gfCNCPoint4[25196] = {X 2.3034, Y 2.3049, Z -6.3333, A 0.000, B 0.000, C 0.000 }
gfCNCPoint4[25197] = {X 2.3034, Y 6.8597, Z -6.3333, A 0.000, B 0.000, C 0.000 }
gfCNCPoint4[25198] = {X 2.4167, Y 6.8824, Z -6.3333, A 0.000, B 0.000, C 0.000 }
gfCNCPoint4[25199] = {X 4.7221, Y 6.0045, Z -6.3333, A 0.000, B 0.000, C 0.000 }
gfCNCPoint4[25200] = {X 7.0996, Y 5.3466, Z -6.3333, A 0.000, B 0.000, C 0.000 }
gfCNCPoint4[25201] = {X 9.5283, Y 4.9145, Z -6.3333, A 0.000, B 0.000, C 0.000 }
gfCNCPoint4[25202] = {X 11.9868, Y 4.7120, Z -6.3333, A 0.000, B 0.000, C 0.000 }
gfCNCPoint4[25203] = {X 14.4535, Y 4.7409, Z -6.3333, A 0.000, B 0.000, C 0.000 }
gfCNCPoint4[25204] = {X 16.9066, Y 5.0009, Z -6.3333, A 0.000, B 0.000, C 0.000 }
gfCNCPoint4[25205] = {X 18.9210, Y 5.4155, Z -6.3333, A 0.000, B 0.000, C 0.000 }
gfCNCPoint4[25206] = {X 20.8820, Y 6.0355, Z -6.3333, A 0.000, B 0.000, C 0.000 }
gfCNCPoint4[25207] = {X 22.7686, Y 6.8543, Z -6.3333, A 0.000, B 0.000, C 0.000 }
gfCNCPoint4[25208] = {X 24.4892, Y 7.8180, Z -6.3333, A 0.000, B 0.000, C 0.000 }
gfCNCPoint4[25209] = {X 26.1061, Y 8.9471, Z -6.3333, A 0.000, B 0.000, C 0.000 }
gfCNCPoint4[25210] = {X 27.4004, Y 10.0775, Z -6.3333, A 0.000, B 0.000, C 0.000 }
gfCNCPoint4[25211] = {X 28.5615, Y 11.3443, Z -6.3333, A 0.000, B 0.000, C 0.000 }
gfCNCPoint4[25212] = {X 29.5750, Y 12.7320, Z -6.3333, A 0.000, B 0.000, C 0.000 }
gfCNCPoint4[25213] = {X 30.4284, Y 14.2234, Z -6.3333, A 0.000, B 0.000, C 0.000 }
gfCNCPoint4[25214] = {X 31.1113, Y 15.8003, Z -6.3333, A 0.000, B 0.000, C 0.000 }
gfCNCPoint4[25215] = {X 31.6710, Y 17.7360, Z -6.3333, A 0.000, B 0.000, C 0.000 }
gfCNCPoint4[25216] = {X 32.0043, Y 19.7232, Z -6.3333, A 0.000, B 0.000, C 0.000 }
gfCNCPoint4[25217] = {X 32.1066, Y 21.7356, Z -6.3333, A 0.000, B 0.000, C 0.000 }
gfCNCPoint4[25218] = {X 31.9766, Y 23.7463, Z -6.3333, A 0.000, B 0.000, C 0.000 }
gfCNCPoint4[25219] = {X 31.6161, Y 25.7288, Z -6.3333, A 0.000, B 0.000, C 0.000 }
gfCNCPoint4[25220] = {X 31.1971, Y 27.1578, Z -6.3333, A 0.000, B 0.000, C 0.000 }
gfCNCPoint4[25221] = {X 30.6305, Y 28.5350, Z -6.3333, A 0.000, B 0.000, C 0.000 }
gfCNCPoint4[25222] = {X 29.9224, Y 29.8451, Z -6.3333, A 0.000, B 0.000, C 0.000 }
gfCNCPoint4[25223] = {X 29.0809, Y 31.0736, Z -6.3333, A 0.000, B 0.000, C 0.000 }
gfCNCPoint4[25224] = {X 29.6386, Y 31.7921, Z -6.3333, A 0.000, B 0.000, C 0.000 }
gfCNCPoint4[25225] = {X 30.0955, Y 32.5786, Z -6.3333, A 0.000, B 0.000, C 0.000 }
gfCNCPoint4[25226] = {X 33.1423, Y 38.8726, Z -6.3333, A 0.000, B 0.000, C 0.000 }
gfCNCPoint4[25227] = {X 33.5391, Y 39.8957, Z -6.3333, A 0.000, B 0.000, C 0.000 }
gfCNCPoint4[25228] = {X 33.7662, Y 40.9694, Z -6.3333, A 0.000, B 0.000, C 0.000 }
gfCNCPoint4[25229] = {X 33.8177, Y 42.0656, Z -6.3333, A 0.000, B 0.000, C 0.000 }
gfCNCPoint4[25230] = {X 33.7164, Y 43.0266, Z -6.3333, A 0.000, B 0.000, C 0.000 }
gfCNCPoint4[25231] = {X 33.4799, Y 43.9636, Z -6.3333, A 0.000, B 0.000, C 0.000 }
gfCNCPoint4[25232] = {X 33.1103, Y 44.8630, Z -6.3333, A 0.000, B 0.000, C 0.000 }
gfCNCPoint4[25233] = {X 32.6161, Y 45.7005, Z -6.3333, A 0.000, B 0.000, C 0.000 }
gfCNCPoint4[25234] = {X 32.0075, Y 46.4590, Z -6.3333, A 0.000, B 0.000, C 0.000 }
gfCNCPoint4[25235] = {X 31.2970, Y 47.1229, Z -6.3333, A 0.000, B 0.000, C 0.000 }
gfCNCPoint4[25236] = {X 30.7609, Y 47.5564, Z -6.3333, A 0.000, B 0.000, C 0.000 }
gfCNCPoint4[25237] = {X 29.8550, Y 48.1752, Z -6.3333, A 0.000, B 0.000, C 0.000 }
gfCNCPoint4[25238] = {X 28.8614, Y 48.6406, Z -6.3333, A 0.000, B 0.000, C 0.000 }
gfCNCPoint4[25239] = {X 27.8061, Y 48.9404, Z -6.3333, A 0.000, B 0.000, C 0.000 }
gfCNCPoint4[25240] = {X 26.7162, Y 49.0669, Z -6.3333, A 0.000, B 0.000, C 0.000 }
gfCNCPoint4[25241] = {X 25.6202, Y 49.0168, Z -6.3333, A 0.000, B 0.000, C 0.000 }
gfCNCPoint4[25242] = {X 23.9293, Y 49.8556, Z -6.3333, A 0.000, B 0.000, C 0.000 }
gfCNCPoint4[25243] = {X 22.1916, Y 50.5926, Z -6.3333, A 0.000, B 0.000, C 0.000 }
gfCNCPoint4[25244] = {X 20.4133, Y 51.2255, Z -6.3333, A 0.000, B 0.000, C 0.000 }
gfCNCPoint4[25245] = {X 18.2641, Y 51.8314, Z -6.3333, A 0.000, B 0.000, C 0.000 }
gfCNCPoint4[25246] = {X 16.0697, Y 52.2450, Z -6.3333, A 0.000, B 0.000, C 0.000 }
gfCNCPoint4[25247] = {X 13.8474, Y 52.4629, Z -6.3333, A 0.000, B 0.000, C 0.000 }
gfCNCPoint4[25248] = {X 11.6145, Y 52.4835, Z -6.3333, A 0.000, B 0.000, C 0.000 }
gfCNCPoint4[25249] = {X 9.3885, Y 52.3066, Z -6.3333, A 0.000, B 0.000, C 0.000 }
gfCNCPoint4[25250] = {X 7.1868, Y 51.9336, Z -6.3333, A 0.000, B 0.000, C 0.000 }
gfCNCPoint4[25251] = {X 6.2986, Y 51.7232, Z -6.3333, A 0.000, B 0.000, C 0.000 }
gfCNCPoint4[25252] = {X 5.4214, Y 51.4709, Z -6.3333, A 0.000, B 0.000, C 0.000 }
gfCNCPoint4[25253] = {X 3.8340, Y 50.8954, Z -6.3333, A 0.000, B 0.000, C 0.000 }
gfCNCPoint4[25254] = {X 2.3034, Y 50.1826, Z -6.3333, A 0.000, B 0.000, C 0.000 }
gfCNCPoint4[25255] = {X 2.3034, Y 97.6951, Z -6.3333, A 0.000, B 0.000, C 0.000 }
gfCNCPoint4[25256] = {X 120.1200, Y 97.6951, Z -6.3333, A 0.000, B 0.000, C 0.000 }
gfCNCPoint4[25257] = {X 120.1200, Y 97.0659, Z -6.3333, A 0.000, B 0.000, C 0.000 }
gfCNCPoint4[25258] = {X 120.2337, Y 96.0185, Z -6.3333, A 0.000, B 0.000, C 0.000 }
gfCNCPoint4[25259] = {X 120.5696, Y 95.0199, Z -6.3333, A 0.000, B 0.000, C 0.000 }
gfCNCPoint4[25260] = {X 121.1121, Y 94.1166, Z -6.3333, A 0.000, B 0.000, C 0.000 }
gfCNCPoint4[25261] = {X 121.8357, Y 93.3509, Z -6.3333, A 0.000, B 0.000, C 0.000 }
gfCNCPoint4[25262] = {X 122.7069, Y 92.7583, Z -6.3333, A 0.000, B 0.000, C 0.000 }
gfCNCPoint4[25263] = {X 123.6849, Y 92.3665, Z -6.3333, A 0.000, B 0.000, C 0.000 }
gfCNCPoint4[25264] = {X 124.7243, Y 92.1937, Z -6.3333, A 0.000, B 0.000, C 0.000 }
gfCNCPoint4[25265] = {X 124.7845, Y 92.1782, Z -6.3333, A 0.000, B 0.000, C 0.000 }
gfCNCPoint4[25266] = {X 124.8456, Y 92.1669, Z -6.3333, A 0.000, B 0.000, C 0.000 }
gfCNCPoint4[25267] = {X 125.3649, Y 92.0898, Z -6.3333, A 0.000, B 0.000, C 0.000 }
gfCNCPoint4[25268] = {X 126.0997, Y 91.9688, Z -6.3333, A 0.000, B 0.000, C 0.000 }
gfCNCPoint4[25269] = {X 126.8253, Y 91.8014, Z -6.3333, A 0.000, B 0.000, C 0.000 }
gfCNCPoint4[25270] = {X 127.9746, Y 90.7110, Z -6.3333, A 0.000, B 0.000, C 0.000 }
gfCNCPoint4[25271] = {X 129.0653, Y 89.5619, Z -6.3333, A 0.000, B 0.000, C 0.000 }
gfCNCPoint4[25272] = {X 154.9458, Y 61.1416, Z -6.3333, A 0.000, B 0.000, C 0.000 }
gfCNCPoint4[25273] = {X 154.6591, Y 60.4492, Z -6.3333, A 0.000, B 0.000, C 0.000 }
gfCNCPoint4[25274] = {X 154.4818, Y 59.7211, Z -6.3333, A 0.000, B 0.000, C 0.000 }
gfCNCPoint4[25275] = {X 154.4181, Y 58.9744, Z -6.3333, A 0.000, B 0.000, C 0.000 }
gfCNCPoint4[25276] = {X 154.4180, Y 58.0000, Z -6.3333, A 0.000, B 0.000, C 0.000 }
gfCNCPoint4[25277] = {X 154.5117, Y 57.0480, Z -6.3333, A 0.000, B 0.000, C 0.000 }
gfCNCPoint4[25278] = {X 154.7894, Y 56.1325, Z -6.3333, A 0.000, B 0.000, C 0.000 }
gfCNCPoint4[25279] = {X 155.2404, Y 55.2888, Z -6.3333, A 0.000, B 0.000, C 0.000 }
gfCNCPoint4[25280] = {X 155.8473, Y 54.5493, Z -6.3333, A 0.000, B 0.000, C 0.000 }
gfCNCPoint4[25281] = {X 156.5868, Y 53.9424, Z -6.3333, A 0.000, B 0.000, C 0.000 }
gfCNCPoint4[25282] = {X 157.4305, Y 53.4915, Z -6.3333, A 0.000, B 0.000, C 0.000 }
gfCNCPoint4[25283] = {X 158.3459, Y 53.2138, Z -6.3333, A 0.000, B 0.000, C 0.000 }
gfCNCPoint4[25284] = {X 159.2980, Y 53.1200, Z -6.3333, A 0.000, B 0.000, C 0.000 }
gfCNCPoint4[25285] = {X 178.5335, Y 53.1200, Z -6.3333, A 0.000, B 0.000, C 0.000 }
gfCNCPoint4[25286] = {X 179.4855, Y 53.2138, Z -6.3333, A 0.000, B 0.000, C 0.000 }
gfCNCPoint4[25287] = {X 180.4010, Y 53.4915, Z -6.3333, A 0.000, B 0.000, C 0.000 }
gfCNCPoint4[25288] = {X 181.2447, Y 53.9424, Z -6.3333, A 0.000, B 0.000, C 0.000 }
gfCNCPoint4[25289] = {X 181.9842, Y 54.5493, Z -6.3333, A 0.000, B 0.000, C 0.000 }
gfCNCPoint4[25290] = {X 182.5911, Y 55.2888, Z -6.3333, A 0.000, B 0.000, C 0.000 }
gfCNCPoint4[25291] = {X 183.0420, Y 56.1325, Z -6.3333, A 0.000, B 0.000, C 0.000 }
gfCNCPoint4[25292] = {X 183.3197, Y 57.0480, Z -6.3333, A 0.000, B 0.000, C 0.000 }
gfCNCPoint4[25293] = {X 183.4135, Y 58.0000, Z -6.3333, A 0.000, B 0.000, C 0.000 }
gfCNCPoint4[25294] = {X 183.4133, Y 58.9744, Z -6.3333, A 0.000, B 0.000, C 0.000 }
gfCNCPoint4[25295] = {X 183.3512, Y 59.7111, Z -6.3333, A 0.000, B 0.000, C 0.000 }
gfCNCPoint4[25296] = {X 183.1786, Y 60.4299, Z -6.3333, A 0.000, B 0.000, C 0.000 }
gfCNCPoint4[25297] = {X 182.8993, Y 61.1144, Z -6.3333, A 0.000, B 0.000, C 0.000 }
gfCNCPoint4[25298] = {X 209.8925, Y 90.5760, Z -6.3333, A 0.000, B 0.000, C 0.000 }
gfCNCPoint4[25299] = {X 210.5203, Y 91.2130, Z -6.3333, A 0.000, B 0.000, C 0.000 }
gfCNCPoint4[25300] = {X 211.1928, Y 91.8026, Z -6.3333, A 0.000, B 0.000, C 0.000 }
gfCNCPoint4[25301] = {X 211.3593, Y 91.9073, Z -6.3333, A 0.000, B 0.000, C 0.000 }
gfCNCPoint4[25302] = {X 211.5461, Y 91.9686, Z -6.3333, A 0.000, B 0.000, C 0.000 }
gfCNCPoint4[25303] = {X 212.2018, Y 92.1088, Z -6.3333, A 0.000, B 0.000, C 0.000 }
gfCNCPoint4[25304] = {X 213.4084, Y 92.2608, Z -6.3333, A 0.000, B 0.000, C 0.000 }
gfCNCPoint4[25305] = {X 214.4425, Y 92.1746, Z -6.3333, A 0.000, B 0.000, C 0.000 }
gfCNCPoint4[25306] = {X 215.4785, Y 92.1156, Z -6.3333, A 0.000, B 0.000, C 0.000 }
gfCNCPoint4[25307] = {X 216.0524, Y 92.0560, Z -6.3333, A 0.000, B 0.000, C 0.000 }
gfCNCPoint4[25308] = {X 216.6053, Y 91.8908, Z -6.3333, A 0.000, B 0.000, C 0.000 }
gfCNCPoint4[25309] = {X 217.1178, Y 91.6256, Z -6.3333, A 0.000, B 0.000, C 0.000 }
gfCNCPoint4[25310] = {X 244.6002, Y 74.0196, Z -6.3333, A 0.000, B 0.000, C 0.000 }
gfCNCPoint4[25311] = {X 221.4279, Y 64.9264, Z -6.3333, A 0.000, B 0.000, C 0.000 }
gfCNCPoint4[25312] = {X 219.7199, Y 64.3542, Z -6.3333, A 0.000, B 0.000, C 0.000 }
gfCNCPoint4[25313] = {X 217.9577, Y 63.9809, Z -6.3333, A 0.000, B 0.000, C 0.000 }
gfCNCPoint4[25314] = {X 216.1644, Y 63.8112, Z -6.3333, A 0.000, B 0.000, C 0.000 }
gfCNCPoint4[25315] = {X 215.1119, Y 63.6594, Z -6.3333, A 0.000, B 0.000, C 0.000 }
gfCNCPoint4[25316] = {X 214.1172, Y 63.2831, Z -6.3333, A 0.000, B 0.000, C 0.000 }
gfCNCPoint4[25317] = {X 213.2277, Y 62.7004, Z -6.3333, A 0.000, B 0.000, C 0.000 }
gfCNCPoint4[25318] = {X 212.4855, Y 61.9388, Z -6.3333, A 0.000, B 0.000, C 0.000 }
gfCNCPoint4[25319] = {X 211.9260, Y 61.0345, Z -6.3333, A 0.000, B 0.000, C 0.000 }
gfCNCPoint4[25320] = {X 211.5756, Y 60.0305, Z -6.3333, A 0.000, B 0.000, C 0.000 }
gfCNCPoint4[25321] = {X 211.4510, Y 58.9744, Z -6.3333, A 0.000, B 0.000, C 0.000 }
gfCNCPoint4[25322] = {X 211.4508, Y 58.0000, Z -6.3333, A 0.000, B 0.000, C 0.000 }
gfCNCPoint4[25323] = {X 211.5446, Y 57.0480, Z -6.3333, A 0.000, B 0.000, C 0.000 }
gfCNCPoint4[25324] = {X 211.8223, Y 56.1325, Z -6.3333, A 0.000, B 0.000, C 0.000 }
gfCNCPoint4[25325] = {X 212.2732, Y 55.2888, Z -6.3333, A 0.000, B 0.000, C 0.000 }
gfCNCPoint4[25326] = {X 212.8801, Y 54.5493, Z -6.3333, A 0.000, B 0.000, C 0.000 }
gfCNCPoint4[25327] = {X 213.6196, Y 53.9424, Z -6.3333, A 0.000, B 0.000, C 0.000 }
gfCNCPoint4[25328] = {X 214.4633, Y 53.4915, Z -6.3333, A 0.000, B 0.000, C 0.000 }
gfCNCPoint4[25329] = {X 215.3788, Y 53.2138, Z -6.3333, A 0.000, B 0.000, C 0.000 }
gfCNCPoint4[25330] = {X 216.3308, Y 53.1200, Z -6.3333, A 0.000, B 0.000, C 0.000 }
gfCNCPoint4[25331] = {X 237.2617, Y 53.1200, Z -6.3333, A 0.000, B 0.000, C 0.000 }
gfCNCPoint4[25332] = {X 238.3265, Y 53.2376, Z -6.3333, A 0.000, B 0.000, C 0.000 }
gfCNCPoint4[25333] = {X 239.3399, Y 53.5846, Z -6.3333, A 0.000, B 0.000, C 0.000 }
gfCNCPoint4[25334] = {X 240.2532, Y 54.1445, Z -6.3333, A 0.000, B 0.000, C 0.000 }
gfCNCPoint4[25335] = {X 241.0224, Y 54.8901, Z -6.3333, A 0.000, B 0.000, C 0.000 }
gfCNCPoint4[25336] = {X 241.6103, Y 55.7855, Z -6.3333, A 0.000, B 0.000, C 0.000 }
gfCNCPoint4[25337] = {X 241.9887, Y 56.7877, Z -6.3333, A 0.000, B 0.000, C 0.000 }
gfCNCPoint4[25338] = {X 242.1393, Y 57.8483, Z -6.3333, A 0.000, B 0.000, C 0.000 }
gfCNCPoint4[25339] = {X 248.3220, Y 60.2592, Z -6.3333, A 0.000, B 0.000, C 0.000 }
gfCNCPoint4[25340] = {X 275.0721, Y 70.8768, Z -6.3333, A 0.000, B 0.000, C 0.000 }
gfCNCPoint4[25341] = {X 275.0718, Y 63.6740, Z -6.3333, A 0.000, B 0.000, C 0.000 }
gfCNCPoint4[25342] = {X 274.0637, Y 63.3055, Z -6.3333, A 0.000, B 0.000, C 0.000 }
gfCNCPoint4[25343] = {X 273.1605, Y 62.7256, Z -6.3333, A 0.000, B 0.000, C 0.000 }
gfCNCPoint4[25344] = {X 272.4059, Y 61.9623, Z -6.3333, A 0.000, B 0.000, C 0.000 }
gfCNCPoint4[25345] = {X 271.8365, Y 61.0525, Z -6.3333, A 0.000, B 0.000, C 0.000 }
gfCNCPoint4[25346] = {X 271.4797, Y 60.0402, Z -6.3333, A 0.000, B 0.000, C 0.000 }
gfCNCPoint4[25347] = {X 271.3529, Y 58.9744, Z -6.3333, A 0.000, B 0.000, C 0.000 }
gfCNCPoint4[25348] = {X 271.3527, Y 58.0000, Z -6.3333, A 0.000, B 0.000, C 0.000 }
gfCNCPoint4[25349] = {X 271.4465, Y 57.0480, Z -6.3333, A 0.000, B 0.000, C 0.000 }
gfCNCPoint4[25350] = {X 271.7242, Y 56.1325, Z -6.3333, A 0.000, B 0.000, C 0.000 }
gfCNCPoint4[25351] = {X 272.1751, Y 55.2888, Z -6.3333, A 0.000, B 0.000, C 0.000 }
gfCNCPoint4[25352] = {X 272.7820, Y 54.5493, Z -6.3333, A 0.000, B 0.000, C 0.000 }
gfCNCPoint4[25353] = {X 273.5215, Y 53.9424, Z -6.3333, A 0.000, B 0.000, C 0.000 }
gfCNCPoint4[25354] = {X 274.3652, Y 53.4915, Z -6.3333, A 0.000, B 0.000, C 0.000 }
gfCNCPoint4[25355] = {X 275.2806, Y 53.2138, Z -6.3333, A 0.000, B 0.000, C 0.000 }
gfCNCPoint4[25356] = {X 276.2327, Y 53.1200, Z -6.3333, A 0.000, B 0.000, C 0.000 }
gfCNCPoint4[25357] = {X 292.7731, Y 53.1200, Z -6.3333, A 0.000, B 0.000, C 0.000 }
gfCNCPoint4[25358] = {X 293.7251, Y 53.2138, Z -6.3333, A 0.000, B 0.000, C 0.000 }
gfCNCPoint4[25359] = {X 294.6406, Y 53.4915, Z -6.3333, A 0.000, B 0.000, C 0.000 }
gfCNCPoint4[25360] = {X 295.4843, Y 53.9424, Z -6.3333, A 0.000, B 0.000, C 0.000 }
gfCNCPoint4[25361] = {X 296.2238, Y 54.5493, Z -6.3333, A 0.000, B 0.000, C 0.000 }
gfCNCPoint4[25362] = {X 296.8307, Y 55.2888, Z -6.3333, A 0.000, B 0.000, C 0.000 }
gfCNCPoint4[25363] = {X 297.2816, Y 56.1325, Z -6.3333, A 0.000, B 0.000, C 0.000 }
gfCNCPoint4[25364] = {X 297.5593, Y 57.0480, Z -6.3333, A 0.000, B 0.000, C 0.000 }
gfCNCPoint4[25365] = {X 297.6531, Y 58.0000, Z -6.3333, A 0.000, B 0.000, C 0.000 }
gfCNCPoint4[25366] = {X 297.6531, Y 58.9365, Z -6.3333, A 0.000, B 0.000, C 0.000 }
gfCNCPoint4[25367] = {X 297.5311, Y 60.0089, Z -6.3333, A 0.000, B 0.000, C 0.000 }
gfCNCPoint4[25368] = {X 297.1771, Y 61.0284, Z -6.3333, A 0.000, B 0.000, C 0.000 }
gfCNCPoint4[25369] = {X 296.6083, Y 61.9457, Z -6.3333, A 0.000, B 0.000, C 0.000 }
gfCNCPoint4[25370] = {X 295.8524, Y 62.7160, Z -6.3333, A 0.000, B 0.000, C 0.000 }
gfCNCPoint4[25371] = {X 294.9461, Y 63.3020, Z -6.3333, A 0.000, B 0.000, C 0.000 }
gfCNCPoint4[25372] = {X 293.9334, Y 63.6753, Z -6.3333, A 0.000, B 0.000, C 0.000 }
gfCNCPoint4[25373] = {X 293.9334, Y 92.3196, Z -6.3333, A 0.000, B 0.000, C 0.000 }
gfCNCPoint4[25374] = {X 294.9453, Y 92.6950, Z -6.3333, A 0.000, B 0.000, C 0.000 }
gfCNCPoint4[25375] = {X 295.8507, Y 93.2824, Z -6.3333, A 0.000, B 0.000, C 0.000 }
gfCNCPoint4[25376] = {X 296.6060, Y 94.0533, Z -6.3333, A 0.000, B 0.000, C 0.000 }
gfCNCPoint4[25377] = {X 297.1747, Y 94.9705, Z -6.3333, A 0.000, B 0.000, C 0.000 }
gfCNCPoint4[25378] = {X 297.5295, Y 95.9897, Z -6.3333, A 0.000, B 0.000, C 0.000 }
gfCNCPoint4[25379] = {X 297.6531, Y 97.0619, Z -6.3333, A 0.000, B 0.000, C 0.000 }
gfCNCPoint4[25380] = {X 297.6531, Y 97.6951, Z -6.3333, A 0.000, B 0.000, C 0.000 }
gfCNCPoint4[25381] = {X 297.1731, Y 97.6951, Z -6.3333, A 0.000, B 0.000, C 0.000 }
gfCNCPoint4[25382] = {X 297.1731, Y 98.0000, Z -6.3333, A 0.000, B 0.000, C 0.000 }
gfCNCPoint4[25383] = {X 297.0628, Y 98.9791, Z -6.3333, A 0.000, B 0.000, C 0.000 }
gfCNCPoint4[25384] = {X 296.7373, Y 99.9091, Z -6.3333, A 0.000, B 0.000, C 0.000 }
gfCNCPoint4[25385] = {X 296.2131, Y 100.7434, Z -6.3333, A 0.000, B 0.000, C 0.000 }
gfCNCPoint4[25386] = {X 295.5164, Y 101.4401, Z -6.3333, A 0.000, B 0.000, C 0.000 }
gfCNCPoint4[25387] = {X 294.6822, Y 101.9643, Z -6.3333, A 0.000, B 0.000, C 0.000 }
gfCNCPoint4[25388] = {X 293.7522, Y 102.2897, Z -6.3333, A 0.000, B 0.000, C 0.000 }
gfCNCPoint4[25389] = {X 292.7731, Y 102.4000, Z -6.3333, A 0.000, B 0.000, C 0.000 }
gfCNCPoint4[25390] = {X 276.2327, Y 102.4000, Z -6.3333, A 0.000, B 0.000, C 0.000 }
gfCNCPoint4[25391] = {X 275.2536, Y 102.2897, Z -6.3333, A 0.000, B 0.000, C 0.000 }
gfCNCPoint4[25392] = {X 274.3236, Y 101.9643, Z -6.3333, A 0.000, B 0.000, C 0.000 }
gfCNCPoint4[25393] = {X 273.4893, Y 101.4401, Z -6.3333, A 0.000, B 0.000, C 0.000 }
gfCNCPoint4[25394] = {X 272.7926, Y 100.7434, Z -6.3333, A 0.000, B 0.000, C 0.000 }
gfCNCPoint4[25395] = {X 272.2684, Y 99.9091, Z -6.3333, A 0.000, B 0.000, C 0.000 }
gfCNCPoint4[25396] = {X 271.9430, Y 98.9791, Z -6.3333, A 0.000, B 0.000, C 0.000 }
gfCNCPoint4[25397] = {X 271.8327, Y 98.0000, Z -6.3333, A 0.000, B 0.000, C 0.000 }
gfCNCPoint4[25398] = {X 271.8329, Y 97.0190, Z -6.3333, A 0.000, B 0.000, C 0.000 }
gfCNCPoint4[25399] = {X 271.9305, Y 96.1432, Z -6.3333, A 0.000, B 0.000, C 0.000 }
gfCNCPoint4[25400] = {X 272.2006, Y 95.3045, Z -6.3333, A 0.000, B 0.000, C 0.000 }
gfCNCPoint4[25401] = {X 272.6325, Y 94.5364, Z -6.3333, A 0.000, B 0.000, C 0.000 }
gfCNCPoint4[25402] = {X 273.2087, Y 93.8698, Z -6.3333, A 0.000, B 0.000, C 0.000 }
gfCNCPoint4[25403] = {X 273.9062, Y 93.3313, Z -6.3333, A 0.000, B 0.000, C 0.000 }
gfCNCPoint4[25404] = {X 274.6970, Y 92.9426, Z -6.3333, A 0.000, B 0.000, C 0.000 }
gfCNCPoint4[25405] = {X 275.5494, Y 92.7193, Z -6.3333, A 0.000, B 0.000, C 0.000 }
gfCNCPoint4[25406] = {X 275.5494, Y 85.6495, Z -6.3333, A 0.000, B 0.000, C 0.000 }
gfCNCPoint4[25407] = {X 262.6483, Y 80.5923, Z -6.3333, A 0.000, B 0.000, C 0.000 }
gfCNCPoint4[25408] = {X 262.3209, Y 80.7990, Z -6.3333, A 0.000, B 0.000, C 0.000 }
gfCNCPoint4[25409] = {X 237.8774, Y 96.6316, Z -6.3333, A 0.000, B 0.000, C 0.000 }
gfCNCPoint4[25410] = {X 237.8798, Y 97.0659, Z -6.3333, A 0.000, B 0.000, C 0.000 }
gfCNCPoint4[25411] = {X 237.8798, Y 98.0000, Z -6.3333, A 0.000, B 0.000, C 0.000 }
gfCNCPoint4[25412] = {X 237.7695, Y 98.9791, Z -6.3333, A 0.000, B 0.000, C 0.000 }
gfCNCPoint4[25413] = {X 237.4440, Y 99.9091, Z -6.3333, A 0.000, B 0.000, C 0.000 }
gfCNCPoint4[25414] = {X 236.9198, Y 100.7434, Z -6.3333, A 0.000, B 0.000, C 0.000 }
gfCNCPoint4[25415] = {X 236.2231, Y 101.4401, Z -6.3333, A 0.000, B 0.000, C 0.000 }
gfCNCPoint4[25416] = {X 235.3889, Y 101.9643, Z -6.3333, A 0.000, B 0.000, C 0.000 }
gfCNCPoint4[25417] = {X 234.4589, Y 102.2897, Z -6.3333, A 0.000, B 0.000, C 0.000 }
gfCNCPoint4[25418] = {X 233.4798, Y 102.4000, Z -6.3333, A 0.000, B 0.000, C 0.000 }
gfCNCPoint4[25419] = {X 214.1790, Y 102.4000, Z -6.3333, A 0.000, B 0.000, C 0.000 }
gfCNCPoint4[25420] = {X 213.7862, Y 102.3824, Z -6.3333, A 0.000, B 0.000, C 0.000 }
gfCNCPoint4[25421] = {X 213.3966, Y 102.3299, Z -6.3333, A 0.000, B 0.000, C 0.000 }
gfCNCPoint4[25422] = {X 213.0069, Y 102.3824, Z -6.3333, A 0.000, B 0.000, C 0.000 }
gfCNCPoint4[25423] = {X 212.6141, Y 102.4000, Z -6.3333, A 0.000, B 0.000, C 0.000 }
gfCNCPoint4[25424] = {X 194.9870, Y 102.4000, Z -6.3333, A 0.000, B 0.000, C 0.000 }
gfCNCPoint4[25425] = {X 194.0079, Y 102.2897, Z -6.3333, A 0.000, B 0.000, C 0.000 }
gfCNCPoint4[25426] = {X 193.0779, Y 101.9643, Z -6.3333, A 0.000, B 0.000, C 0.000 }
gfCNCPoint4[25427] = {X 192.2436, Y 101.4401, Z -6.3333, A 0.000, B 0.000, C 0.000 }
gfCNCPoint4[25428] = {X 191.5469, Y 100.7434, Z -6.3333, A 0.000, B 0.000, C 0.000 }
gfCNCPoint4[25429] = {X 191.0227, Y 99.9091, Z -6.3333, A 0.000, B 0.000, C 0.000 }
gfCNCPoint4[25430] = {X 190.6973, Y 98.9791, Z -6.3333, A 0.000, B 0.000, C 0.000 }
gfCNCPoint4[25431] = {X 190.5870, Y 98.0000, Z -6.3333, A 0.000, B 0.000, C 0.000 }
gfCNCPoint4[25432] = {X 190.5870, Y 97.0659, Z -6.3333, A 0.000, B 0.000, C 0.000 }
gfCNCPoint4[25433] = {X 190.6897, Y 96.1207, Z -6.3333, A 0.000, B 0.000, C 0.000 }
gfCNCPoint4[25434] = {X 190.9931, Y 95.2196, Z -6.3333, A 0.000, B 0.000, C 0.000 }
gfCNCPoint4[25435] = {X 191.4830, Y 94.4047, Z -6.3333, A 0.000, B 0.000, C 0.000 }
gfCNCPoint4[25436] = {X 188.5295, Y 91.1802, Z -6.3333, A 0.000, B 0.000, C 0.000 }
gfCNCPoint4[25437] = {X 150.1254, Y 91.1802, Z -6.3333, A 0.000, B 0.000, C 0.000 }
gfCNCPoint4[25438] = {X 147.2501, Y 94.3657, Z -6.3333, A 0.000, B 0.000, C 0.000 }
gfCNCPoint4[25439] = {X 147.7563, Y 95.1900, Z -6.3333, A 0.000, B 0.000, C 0.000 }
gfCNCPoint4[25440] = {X 148.0710, Y 96.1048, Z -6.3333, A 0.000, B 0.000, C 0.000 }
gfCNCPoint4[25441] = {X 148.1791, Y 97.0660, Z -6.3333, A 0.000, B 0.000, C 0.000 }
gfCNCPoint4[25442] = {X 148.1791, Y 98.0000, Z -6.3333, A 0.000, B 0.000, C 0.000 }
gfCNCPoint4[25443] = {X 148.0688, Y 98.9791, Z -6.3333, A 0.000, B 0.000, C 0.000 }
gfCNCPoint4[25444] = {X 147.7434, Y 99.9091, Z -6.3333, A 0.000, B 0.000, C 0.000 }
gfCNCPoint4[25445] = {X 147.2192, Y 100.7434, Z -6.3333, A 0.000, B 0.000, C 0.000 }
gfCNCPoint4[25446] = {X 146.5225, Y 101.4401, Z -6.3333, A 0.000, B 0.000, C 0.000 }
gfCNCPoint4[25447] = {X 145.6882, Y 101.9643, Z -6.3333, A 0.000, B 0.000, C 0.000 }
gfCNCPoint4[25448] = {X 144.7582, Y 102.2897, Z -6.3333, A 0.000, B 0.000, C 0.000 }
gfCNCPoint4[25449] = {X 143.7791, Y 102.4000, Z -6.3333, A 0.000, B 0.000, C 0.000 }
gfCNCPoint4[25450] = {X 125.0000, Y 102.4000, Z -6.3333, A 0.000, B 0.000, C 0.000 }
gfCNCPoint4[25451] = {X 124.0209, Y 102.2897, Z -6.3333, A 0.000, B 0.000, C 0.000 }
gfCNCPoint4[25452] = {X 123.0909, Y 101.9643, Z -6.3333, A 0.000, B 0.000, C 0.000 }
gfCNCPoint4[25453] = {X 122.2566, Y 101.4401, Z -6.3333, A 0.000, B 0.000, C 0.000 }
gfCNCPoint4[25454] = {X 121.5599, Y 100.7434, Z -6.3333, A 0.000, B 0.000, C 0.000 }
gfCNCPoint4[25455] = {X 121.0357, Y 99.9091, Z -6.3333, A 0.000, B 0.000, C 0.000 }
gfCNCPoint4[25456] = {X 120.7103, Y 98.9791, Z -6.3333, A 0.000, B 0.000, C 0.000 }
gfCNCPoint4[25457] = {X 120.6000, Y 98.0000, Z -6.3333, A 0.000, B 0.000, C 0.000 }
gfCNCPoint4[25458] = {X 120.6000, Y 97.0659, Z -6.3333, A 0.000, B 0.000, C 0.000 }
gfCNCPoint4[25459] = {X 120.7046, Y 96.1124, Z -6.3333, A 0.000, B 0.000, C 0.000 }
gfCNCPoint4[25460] = {X 121.0133, Y 95.2041, Z -6.3333, A 0.000, B 0.000, C 0.000 }
gfCNCPoint4[25461] = {X 121.5116, Y 94.3843, Z -6.3333, A 0.000, B 0.000, C 0.000 }
gfCNCPoint4[25462] = {X 122.1757, Y 93.6921, Z -6.3333, A 0.000, B 0.000, C 0.000 }
gfCNCPoint4[25463] = {X 122.9740, Y 93.1601, Z -6.3333, A 0.000, B 0.000, C 0.000 }
gfCNCPoint4[25464] = {X 123.8686, Y 92.8139, Z -6.3333, A 0.000, B 0.000, C 0.000 }
gfCNCPoint4[25465] = {X 124.8170, Y 92.6697, Z -6.3333, A 0.000, B 0.000, C 0.000 }
gfCNCPoint4[25466] = {X 124.8656, Y 92.6525, Z -6.3333, A 0.000, B 0.000, C 0.000 }
gfCNCPoint4[25467] = {X 124.9160, Y 92.6417, Z -6.3333, A 0.000, B 0.000, C 0.000 }
gfCNCPoint4[25468] = {X 125.4412, Y 92.5638, Z -6.3333, A 0.000, B 0.000, C 0.000 }
gfCNCPoint4[25469] = {X 126.2564, Y 92.4269, Z -6.3333, A 0.000, B 0.000, C 0.000 }
gfCNCPoint4[25470] = {X 127.0606, Y 92.2351, Z -6.3333, A 0.000, B 0.000, C 0.000 }
gfCNCPoint4[25471] = {X 128.2723, Y 91.0921, Z -6.3333, A 0.000, B 0.000, C 0.000 }
gfCNCPoint4[25472] = {X 129.4202, Y 89.8851, Z -6.3333, A 0.000, B 0.000, C 0.000 }
gfCNCPoint4[25473] = {X 155.5325, Y 61.2103, Z -6.3333, A 0.000, B 0.000, C 0.000 }
gfCNCPoint4[25474] = {X 155.1839, Y 60.4943, Z -6.3333, A 0.000, B 0.000, C 0.000 }
gfCNCPoint4[25475] = {X 154.9700, Y 59.7272, Z -6.3333, A 0.000, B 0.000, C 0.000 }
gfCNCPoint4[25476] = {X 154.8980, Y 58.9341, Z -6.3333, A 0.000, B 0.000, C 0.000 }
gfCNCPoint4[25477] = {X 154.8980, Y 58.0000, Z -6.3333, A 0.000, B 0.000, C 0.000 }
gfCNCPoint4[25478] = {X 155.0083, Y 57.0209, Z -6.3333, A 0.000, B 0.000, C 0.000 }
gfCNCPoint4[25479] = {X 155.3337, Y 56.0909, Z -6.3333, A 0.000, B 0.000, C 0.000 }
gfCNCPoint4[25480] = {X 155.8579, Y 55.2566, Z -6.3333, A 0.000, B 0.000, C 0.000 }
gfCNCPoint4[25481] = {X 156.5546, Y 54.5599, Z -6.3333, A 0.000, B 0.000, C 0.000 }
gfCNCPoint4[25482] = {X 157.3889, Y 54.0357, Z -6.3333, A 0.000, B 0.000, C 0.000 }
gfCNCPoint4[25483] = {X 158.3189, Y 53.7103, Z -6.3333, A 0.000, B 0.000, C 0.000 }
gfCNCPoint4[25484] = {X 159.2980, Y 53.6000, Z -6.3333, A 0.000, B 0.000, C 0.000 }
gfCNCPoint4[25485] = {X 178.5335, Y 53.6000, Z -6.3333, A 0.000, B 0.000, C 0.000 }
gfCNCPoint4[25486] = {X 179.5126, Y 53.7103, Z -6.3333, A 0.000, B 0.000, C 0.000 }
gfCNCPoint4[25487] = {X 180.4426, Y 54.0357, Z -6.3333, A 0.000, B 0.000, C 0.000 }
gfCNCPoint4[25488] = {X 181.2769, Y 54.5599, Z -6.3333, A 0.000, B 0.000, C 0.000 }
gfCNCPoint4[25489] = {X 181.9736, Y 55.2566, Z -6.3333, A 0.000, B 0.000, C 0.000 }
gfCNCPoint4[25490] = {X 182.4978, Y 56.0909, Z -6.3333, A 0.000, B 0.000, C 0.000 }
gfCNCPoint4[25491] = {X 182.8232, Y 57.0209, Z -6.3333, A 0.000, B 0.000, C 0.000 }
gfCNCPoint4[25492] = {X 182.9335, Y 58.0000, Z -6.3333, A 0.000, B 0.000, C 0.000 }
gfCNCPoint4[25493] = {X 182.9334, Y 58.9704, Z -6.3333, A 0.000, B 0.000, C 0.000 }
gfCNCPoint4[25494] = {X 182.8588, Y 59.7416, Z -6.3333, A 0.000, B 0.000, C 0.000 }
gfCNCPoint4[25495] = {X 182.6501, Y 60.4878, Z -6.3333, A 0.000, B 0.000, C 0.000 }
gfCNCPoint4[25496] = {X 182.3137, Y 61.1858, Z -6.3333, A 0.000, B 0.000, C 0.000 }
gfCNCPoint4[25497] = {X 209.5386, Y 90.9003, Z -6.3333, A 0.000, B 0.000, C 0.000 }
gfCNCPoint4[25498] = {X 210.1910, Y 91.5622, Z -6.3333, A 0.000, B 0.000, C 0.000 }
gfCNCPoint4[25499] = {X 210.8898, Y 92.1748, Z -6.3333, A 0.000, B 0.000, C 0.000 }
gfCNCPoint4[25500] = {X 211.1518, Y 92.3401, Z -6.3333, A 0.000, B 0.000, C 0.000 }
gfCNCPoint4[25501] = {X 211.4457, Y 92.4380, Z -6.3333, A 0.000, B 0.000, C 0.000 }
gfCNCPoint4[25502] = {X 212.1215, Y 92.5825, Z -6.3333, A 0.000, B 0.000, C 0.000 }
gfCNCPoint4[25503] = {X 213.4016, Y 92.7437, Z -6.3333, A 0.000, B 0.000, C 0.000 }
gfCNCPoint4[25504] = {X 214.4548, Y 92.6550, Z -6.3333, A 0.000, B 0.000, C 0.000 }
gfCNCPoint4[25505] = {X 215.5100, Y 92.5948, Z -6.3333, A 0.000, B 0.000, C 0.000 }
gfCNCPoint4[25506] = {X 216.1641, Y 92.5229, Z -6.3333, A 0.000, B 0.000, C 0.000 }
gfCNCPoint4[25507] = {X 216.7938, Y 92.3322, Z -6.3333, A 0.000, B 0.000, C 0.000 }
gfCNCPoint4[25508] = {X 217.3777, Y 92.0291, Z -6.3333, A 0.000, B 0.000, C 0.000 }
gfCNCPoint4[25509] = {X 222.9188, Y 88.4532, Z -6.3333, A 0.000, B 0.000, C 0.000 }
gfCNCPoint4[25510] = {X 245.6521, Y 73.9168, Z -6.3333, A 0.000, B 0.000, C 0.000 }
gfCNCPoint4[25511] = {X 221.6009, Y 64.4787, Z -6.3333, A 0.000, B 0.000, C 0.000 }
gfCNCPoint4[25512] = {X 219.8422, Y 63.8901, Z -6.3333, A 0.000, B 0.000, C 0.000 }
gfCNCPoint4[25513] = {X 218.0279, Y 63.5060, Z -6.3333, A 0.000, B 0.000, C 0.000 }
gfCNCPoint4[25514] = {X 216.1815, Y 63.3315, Z -6.3333, A 0.000, B 0.000, C 0.000 }
gfCNCPoint4[25515] = {X 215.2274, Y 63.1935, Z -6.3333, A 0.000, B 0.000, C 0.000 }
gfCNCPoint4[25516] = {X 214.3262, Y 62.8509, Z -6.3333, A 0.000, B 0.000, C 0.000 }
gfCNCPoint4[25517] = {X 213.5213, Y 62.3203, Z -6.3333, A 0.000, B 0.000, C 0.000 }
gfCNCPoint4[25518] = {X 212.8512, Y 61.6271, Z -6.3333, A 0.000, B 0.000, C 0.000 }
gfCNCPoint4[25519] = {X 212.3482, Y 60.8046, Z -6.3333, A 0.000, B 0.000, C 0.000 }
gfCNCPoint4[25520] = {X 212.0364, Y 59.8923, Z -6.3333, A 0.000, B 0.000, C 0.000 }
gfCNCPoint4[25521] = {X 211.9308, Y 58.9341, Z -6.3333, A 0.000, B 0.000, C 0.000 }
gfCNCPoint4[25522] = {X 211.9308, Y 58.0000, Z -6.3333, A 0.000, B 0.000, C 0.000 }
gfCNCPoint4[25523] = {X 212.0411, Y 57.0209, Z -6.3333, A 0.000, B 0.000, C 0.000 }
gfCNCPoint4[25524] = {X 212.3665, Y 56.0909, Z -6.3333, A 0.000, B 0.000, C 0.000 }
gfCNCPoint4[25525] = {X 212.8907, Y 55.2566, Z -6.3333, A 0.000, B 0.000, C 0.000 }
gfCNCPoint4[25526] = {X 213.5875, Y 54.5599, Z -6.3333, A 0.000, B 0.000, C 0.000 }
gfCNCPoint4[25527] = {X 214.4217, Y 54.0357, Z -6.3333, A 0.000, B 0.000, C 0.000 }
gfCNCPoint4[25528] = {X 215.3517, Y 53.7103, Z -6.3333, A 0.000, B 0.000, C 0.000 }
gfCNCPoint4[25529] = {X 216.3308, Y 53.6000, Z -6.3333, A 0.000, B 0.000, C 0.000 }
gfCNCPoint4[25530] = {X 237.2617, Y 53.6000, Z -6.3333, A 0.000, B 0.000, C 0.000 }
gfCNCPoint4[25531] = {X 238.2408, Y 53.7103, Z -6.3333, A 0.000, B 0.000, C 0.000 }
gfCNCPoint4[25532] = {X 239.1708, Y 54.0357, Z -6.3333, A 0.000, B 0.000, C 0.000 }
gfCNCPoint4[25533] = {X 240.0050, Y 54.5599, Z -6.3333, A 0.000, B 0.000, C 0.000 }
gfCNCPoint4[25534] = {X 240.7017, Y 55.2566, Z -6.3333, A 0.000, B 0.000, C 0.000 }
gfCNCPoint4[25535] = {X 241.2260, Y 56.0909, Z -6.3333, A 0.000, B 0.000, C 0.000 }
gfCNCPoint4[25536] = {X 241.5514, Y 57.0209, Z -6.3333, A 0.000, B 0.000, C 0.000 }
gfCNCPoint4[25537] = {X 241.6617, Y 58.0000, Z -6.3333, A 0.000, B 0.000, C 0.000 }
gfCNCPoint4[25538] = {X 241.6617, Y 58.1773, Z -6.3333, A 0.000, B 0.000, C 0.000 }
gfCNCPoint4[25539] = {X 248.1449, Y 60.7053, Z -6.3333, A 0.000, B 0.000, C 0.000 }
gfCNCPoint4[25540] = {X 275.5521, Y 71.5837, Z -6.3333, A 0.000, B 0.000, C 0.000 }
gfCNCPoint4[25541] = {X 275.5518, Y 63.2811, Z -6.3333, A 0.000, B 0.000, C 0.000 }
gfCNCPoint4[25542] = {X 274.6927, Y 63.0558, Z -6.3333, A 0.000, B 0.000, C 0.000 }
gfCNCPoint4[25543] = {X 273.8963, Y 62.6625, Z -6.3333, A 0.000, B 0.000, C 0.000 }
gfCNCPoint4[25544] = {X 273.1951, Y 62.1173, Z -6.3333, A 0.000, B 0.000, C 0.000 }
gfCNCPoint4[25545] = {X 272.6177, Y 61.4424, Z -6.3333, A 0.000, B 0.000, C 0.000 }
gfCNCPoint4[25546] = {X 272.1876, Y 60.6653, Z -6.3333, A 0.000, B 0.000, C 0.000 }
gfCNCPoint4[25547] = {X 271.9223, Y 59.8177, Z -6.3333, A 0.000, B 0.000, C 0.000 }
gfCNCPoint4[25548] = {X 271.8327, Y 58.9341, Z -6.3333, A 0.000, B 0.000, C 0.000 }
gfCNCPoint4[25549] = {X 271.8327, Y 58.0000, Z -6.3333, A 0.000, B 0.000, C 0.000 }
gfCNCPoint4[25550] = {X 271.9430, Y 57.0209, Z -6.3333, A 0.000, B 0.000, C 0.000 }
gfCNCPoint4[25551] = {X 272.2684, Y 56.0909, Z -6.3333, A 0.000, B 0.000, C 0.000 }
gfCNCPoint4[25552] = {X 272.7926, Y 55.2566, Z -6.3333, A 0.000, B 0.000, C 0.000 }
gfCNCPoint4[25553] = {X 273.4893, Y 54.5599, Z -6.3333, A 0.000, B 0.000, C 0.000 }
gfCNCPoint4[25554] = {X 274.3236, Y 54.0357, Z -6.3333, A 0.000, B 0.000, C 0.000 }
gfCNCPoint4[25555] = {X 275.2536, Y 53.7103, Z -6.3333, A 0.000, B 0.000, C 0.000 }
gfCNCPoint4[25556] = {X 276.2327, Y 53.6000, Z -6.3333, A 0.000, B 0.000, C 0.000 }
gfCNCPoint4[25557] = {X 292.7731, Y 53.6000, Z -6.3333, A 0.000, B 0.000, C 0.000 }
gfCNCPoint4[25558] = {X 293.7522, Y 53.7103, Z -6.3333, A 0.000, B 0.000, C 0.000 }
gfCNCPoint4[25559] = {X 294.6822, Y 54.0357, Z -6.3333, A 0.000, B 0.000, C 0.000 }
gfCNCPoint4[25560] = {X 295.5164, Y 54.5599, Z -6.3333, A 0.000, B 0.000, C 0.000 }
gfCNCPoint4[25561] = {X 296.2131, Y 55.2566, Z -6.3333, A 0.000, B 0.000, C 0.000 }
gfCNCPoint4[25562] = {X 296.7373, Y 56.0909, Z -6.3333, A 0.000, B 0.000, C 0.000 }
gfCNCPoint4[25563] = {X 297.0628, Y 57.0209, Z -6.3333, A 0.000, B 0.000, C 0.000 }
gfCNCPoint4[25564] = {X 297.1731, Y 58.0000, Z -6.3333, A 0.000, B 0.000, C 0.000 }
gfCNCPoint4[25565] = {X 297.1731, Y 58.9352, Z -6.3333, A 0.000, B 0.000, C 0.000 }
gfCNCPoint4[25566] = {X 297.0813, Y 59.8182, Z -6.3333, A 0.000, B 0.000, C 0.000 }
gfCNCPoint4[25567] = {X 296.8148, Y 60.6650, Z -6.3333, A 0.000, B 0.000, C 0.000 }
gfCNCPoint4[25568] = {X 296.3843, Y 61.4414, Z -6.3333, A 0.000, B 0.000, C 0.000 }
gfCNCPoint4[25569] = {X 295.8072, Y 62.1160, Z -6.3333, A 0.000, B 0.000, C 0.000 }
gfCNCPoint4[25570] = {X 295.1069, Y 62.6616, Z -6.3333, A 0.000, B 0.000, C 0.000 }
gfCNCPoint4[25571] = {X 294.3116, Y 63.0560, Z -6.3333, A 0.000, B 0.000, C 0.000 }
gfCNCPoint4[25572] = {X 293.4534, Y 63.2835, Z -6.3333, A 0.000, B 0.000, C 0.000 }
gfCNCPoint4[25573] = {X 293.4534, Y 92.7102, Z -6.3333, A 0.000, B 0.000, C 0.000 }
gfCNCPoint4[25574] = {X 294.3113, Y 92.9402, Z -6.3333, A 0.000, B 0.000, C 0.000 }
gfCNCPoint4[25575] = {X 295.1061, Y 93.3365, Z -6.3333, A 0.000, B 0.000, C 0.000 }
gfCNCPoint4[25576] = {X 295.8060, Y 93.8834, Z -6.3333, A 0.000, B 0.000, C 0.000 }
gfCNCPoint4[25577] = {X 296.3828, Y 94.5588, Z -6.3333, A 0.000, B 0.000, C 0.000 }
gfCNCPoint4[25578] = {X 296.8133, Y 95.3356, Z -6.3333, A 0.000, B 0.000, C 0.000 }
gfCNCPoint4[25579] = {X 297.0803, Y 96.1827, Z -6.3333, A 0.000, B 0.000, C 0.000 }
gfCNCPoint4[25580] = {X 297.1731, Y 97.0660, Z -6.3333, A 0.000, B 0.000, C 0.000 }
gfCNCPoint4[25581] = {X 297.1731, Y 97.6951, Z -6.3333, A 0.000, B 0.000, C 0.000 }
gfCNCPoint4[25582] = {X 297.6531, Y 97.6951, Z -6.3333, A 0.000, B 0.000, C 0.000 }
gfCNCPoint4[25583] = {X 314.2120, Y 97.6951, Z -6.3333, A 0.000, B 0.000, C 0.000 }
gfCNCPoint4[25584] = {X 313.0146, Y 96.8448, Z -6.3333, A 0.000, B 0.000, C 0.000 }
gfCNCPoint4[25585] = {X 311.8812, Y 95.9108, Z -6.3333, A 0.000, B 0.000, C 0.000 }
gfCNCPoint4[25586] = {X 310.9057, Y 94.9488, Z -6.3333, A 0.000, B 0.000, C 0.000 }
gfCNCPoint4[25587] = {X 310.0414, Y 93.8856, Z -6.3333, A 0.000, B 0.000, C 0.000 }
gfCNCPoint4[25588] = {X 309.2074, Y 92.5709, Z -6.3333, A 0.000, B 0.000, C 0.000 }
gfCNCPoint4[25589] = {X 308.5434, Y 91.1627, Z -6.3333, A 0.000, B 0.000, C 0.000 }
gfCNCPoint4[25590] = {X 308.0599, Y 89.6828, Z -6.3333, A 0.000, B 0.000, C 0.000 }
gfCNCPoint4[25591] = {X 307.7064, Y 88.0129, Z -6.3333, A 0.000, B 0.000, C 0.000 }
gfCNCPoint4[25592] = {X 307.4975, Y 86.3188, Z -6.3333, A 0.000, B 0.000, C 0.000 }
gfCNCPoint4[25593] = {X 307.4347, Y 84.6131, Z -6.3333, A 0.000, B 0.000, C 0.000 }
gfCNCPoint4[25594] = {X 307.4359, Y 63.6741, Z -6.3333, A 0.000, B 0.000, C 0.000 }
gfCNCPoint4[25595] = {X 306.4277, Y 63.3058, Z -6.3333, A 0.000, B 0.000, C 0.000 }
gfCNCPoint4[25596] = {X 305.5243, Y 62.7259, Z -6.3333, A 0.000, B 0.000, C 0.000 }
gfCNCPoint4[25597] = {X 304.7696, Y 61.9625, Z -6.3333, A 0.000, B 0.000, C 0.000 }
gfCNCPoint4[25598] = {X 304.2001, Y 61.0527, Z -6.3333, A 0.000, B 0.000, C 0.000 }
gfCNCPoint4[25599] = {X 303.8433, Y 60.0403, Z -6.3333, A 0.000, B 0.000, C 0.000 }
gfCNCPoint4[25600] = {X 303.7164, Y 58.9744, Z -6.3333, A 0.000, B 0.000, C 0.000 }
gfCNCPoint4[25601] = {X 303.7162, Y 58.0000, Z -6.3333, A 0.000, B 0.000, C 0.000 }
gfCNCPoint4[25602] = {X 303.8100, Y 57.0480, Z -6.3333, A 0.000, B 0.000, C 0.000 }
gfCNCPoint4[25603] = {X 304.0877, Y 56.1325, Z -6.3333, A 0.000, B 0.000, C 0.000 }
gfCNCPoint4[25604] = {X 304.5387, Y 55.2888, Z -6.3333, A 0.000, B 0.000, C 0.000 }
gfCNCPoint4[25605] = {X 305.1455, Y 54.5493, Z -6.3333, A 0.000, B 0.000, C 0.000 }
gfCNCPoint4[25606] = {X 305.8850, Y 53.9424, Z -6.3333, A 0.000, B 0.000, C 0.000 }
gfCNCPoint4[25607] = {X 306.7287, Y 53.4915, Z -6.3333, A 0.000, B 0.000, C 0.000 }
gfCNCPoint4[25608] = {X 307.6442, Y 53.2138, Z -6.3333, A 0.000, B 0.000, C 0.000 }
gfCNCPoint4[25609] = {X 308.5962, Y 53.1200, Z -6.3333, A 0.000, B 0.000, C 0.000 }
gfCNCPoint4[25610] = {X 324.3107, Y 53.1200, Z -6.3333, A 0.000, B 0.000, C 0.000 }
gfCNCPoint4[25611] = {X 325.2627, Y 53.2138, Z -6.3333, A 0.000, B 0.000, C 0.000 }
gfCNCPoint4[25612] = {X 326.1782, Y 53.4915, Z -6.3333, A 0.000, B 0.000, C 0.000 }
gfCNCPoint4[25613] = {X 327.0219, Y 53.9424, Z -6.3333, A 0.000, B 0.000, C 0.000 }
gfCNCPoint4[25614] = {X 327.7614, Y 54.5493, Z -6.3333, A 0.000, B 0.000, C 0.000 }
gfCNCPoint4[25615] = {X 328.3683, Y 55.2888, Z -6.3333, A 0.000, B 0.000, C 0.000 }
gfCNCPoint4[25616] = {X 328.8192, Y 56.1325, Z -6.3333, A 0.000, B 0.000, C 0.000 }
gfCNCPoint4[25617] = {X 329.0969, Y 57.0480, Z -6.3333, A 0.000, B 0.000, C 0.000 }
gfCNCPoint4[25618] = {X 329.1907, Y 58.0000, Z -6.3333, A 0.000, B 0.000, C 0.000 }
gfCNCPoint4[25619] = {X 329.1907, Y 58.9341, Z -6.3333, A 0.000, B 0.000, C 0.000 }
gfCNCPoint4[25620] = {X 329.0674, Y 60.0068, Z -6.3333, A 0.000, B 0.000, C 0.000 }
gfCNCPoint4[25621] = {X 328.7129, Y 61.0267, Z -6.3333, A 0.000, B 0.000, C 0.000 }
gfCNCPoint4[25622] = {X 328.1445, Y 61.9447, Z -6.3333, A 0.000, B 0.000, C 0.000 }
gfCNCPoint4[25623] = {X 327.3894, Y 62.7164, Z -6.3333, A 0.000, B 0.000, C 0.000 }
gfCNCPoint4[25624] = {X 326.4840, Y 63.3048, Z -6.3333, A 0.000, B 0.000, C 0.000 }
gfCNCPoint4[25625] = {X 325.4721, Y 63.6815, Z -6.3333, A 0.000, B 0.000, C 0.000 }
gfCNCPoint4[25626] = {X 325.4739, Y 83.2269, Z -6.3333, A 0.000, B 0.000, C 0.000 }
gfCNCPoint4[25627] = {X 325.4874, Y 84.6073, Z -6.3333, A 0.000, B 0.000, C 0.000 }
gfCNCPoint4[25628] = {X 325.5534, Y 85.7199, Z -6.3333, A 0.000, B 0.000, C 0.000 }
gfCNCPoint4[25629] = {X 325.7427, Y 86.8182, Z -6.3333, A 0.000, B 0.000, C 0.000 }
gfCNCPoint4[25630] = {X 325.8869, Y 86.9523, Z -6.3333, A 0.000, B 0.000, C 0.000 }
gfCNCPoint4[25631] = {X 326.0553, Y 87.0541, Z -6.3333, A 0.000, B 0.000, C 0.000 }
gfCNCPoint4[25632] = {X 326.4846, Y 87.2970, Z -6.3333, A 0.000, B 0.000, C 0.000 }
gfCNCPoint4[25633] = {X 327.8574, Y 87.8648, Z -6.3333, A 0.000, B 0.000, C 0.000 }
gfCNCPoint4[25634] = {X 329.2838, Y 88.2799, Z -6.3333, A 0.000, B 0.000, C 0.000 }
gfCNCPoint4[25635] = {X 331.5313, Y 88.7478, Z -6.3333, A 0.000, B 0.000, C 0.000 }
gfCNCPoint4[25636] = {X 333.7990, Y 89.1048, Z -6.3333, A 0.000, B 0.000, C 0.000 }
gfCNCPoint4[25637] = {X 336.0816, Y 89.3499, Z -6.3333, A 0.000, B 0.000, C 0.000 }
gfCNCPoint4[25638] = {X 340.4337, Y 89.6429, Z -6.3333, A 0.000, B 0.000, C 0.000 }
gfCNCPoint4[25639] = {X 344.7930, Y 89.7962, Z -6.3333, A 0.000, B 0.000, C 0.000 }
gfCNCPoint4[25640] = {X 349.1549, Y 89.8094, Z -6.3333, A 0.000, B 0.000, C 0.000 }
gfCNCPoint4[25641] = {X 353.2889, Y 89.7416, Z -6.3333, A 0.000, B 0.000, C 0.000 }
gfCNCPoint4[25642] = {X 357.4177, Y 89.5237, Z -6.3333, A 0.000, B 0.000, C 0.000 }
gfCNCPoint4[25643] = {X 361.5359, Y 89.1560, Z -6.3333, A 0.000, B 0.000, C 0.000 }
gfCNCPoint4[25644] = {X 363.5861, Y 88.8731, Z -6.3333, A 0.000, B 0.000, C 0.000 }
gfCNCPoint4[25645] = {X 365.6175, Y 88.4771, Z -6.3333, A 0.000, B 0.000, C 0.000 }
gfCNCPoint4[25646] = {X 367.6239, Y 87.9691, Z -6.3333, A 0.000, B 0.000, C 0.000 }
gfCNCPoint4[25647] = {X 368.9175, Y 87.4944, Z -6.3333, A 0.000, B 0.000, C 0.000 }
gfCNCPoint4[25648] = {X 370.1133, Y 86.8095, Z -6.3333, A 0.000, B 0.000, C 0.000 }
gfCNCPoint4[25649] = {X 370.2978, Y 85.3242, Z -6.3333, A 0.000, B 0.000, C 0.000 }
gfCNCPoint4[25650] = {X 370.3594, Y 83.8287, Z -6.3333, A 0.000, B 0.000, C 0.000 }
gfCNCPoint4[25651] = {X 370.3582, Y 63.6739, Z -6.3333, A 0.000, B 0.000, C 0.000 }
gfCNCPoint4[25652] = {X 369.3501, Y 63.3055, Z -6.3333, A 0.000, B 0.000, C 0.000 }
gfCNCPoint4[25653] = {X 368.4470, Y 62.7255, Z -6.3333, A 0.000, B 0.000, C 0.000 }
gfCNCPoint4[25654] = {X 367.6924, Y 61.9622, Z -6.3333, A 0.000, B 0.000, C 0.000 }
gfCNCPoint4[25655] = {X 367.1230, Y 61.0524, Z -6.3333, A 0.000, B 0.000, C 0.000 }
gfCNCPoint4[25656] = {X 366.7663, Y 60.0401, Z -6.3333, A 0.000, B 0.000, C 0.000 }
gfCNCPoint4[25657] = {X 366.6394, Y 58.9744, Z -6.3333, A 0.000, B 0.000, C 0.000 }
gfCNCPoint4[25658] = {X 366.6393, Y 58.0000, Z -6.3333, A 0.000, B 0.000, C 0.000 }
gfCNCPoint4[25659] = {X 366.7331, Y 57.0480, Z -6.3333, A 0.000, B 0.000, C 0.000 }
gfCNCPoint4[25660] = {X 367.0108, Y 56.1325, Z -6.3333, A 0.000, B 0.000, C 0.000 }
gfCNCPoint4[25661] = {X 367.4617, Y 55.2888, Z -6.3333, A 0.000, B 0.000, C 0.000 }
gfCNCPoint4[25662] = {X 368.0686, Y 54.5493, Z -6.3333, A 0.000, B 0.000, C 0.000 }
gfCNCPoint4[25663] = {X 368.8081, Y 53.9424, Z -6.3333, A 0.000, B 0.000, C 0.000 }
gfCNCPoint4[25664] = {X 369.6518, Y 53.4915, Z -6.3333, A 0.000, B 0.000, C 0.000 }
gfCNCPoint4[25665] = {X 370.5672, Y 53.2138, Z -6.3333, A 0.000, B 0.000, C 0.000 }
gfCNCPoint4[25666] = {X 371.5193, Y 53.1200, Z -6.3333, A 0.000, B 0.000, C 0.000 }
gfCNCPoint4[25667] = {X 388.0597, Y 53.1200, Z -6.3333, A 0.000, B 0.000, C 0.000 }
gfCNCPoint4[25668] = {X 389.0355, Y 53.2186, Z -6.3333, A 0.000, B 0.000, C 0.000 }
gfCNCPoint4[25669] = {X 389.9719, Y 53.5102, Z -6.3333, A 0.000, B 0.000, C 0.000 }
gfCNCPoint4[25670] = {X 390.8310, Y 53.9833, Z -6.3333, A 0.000, B 0.000, C 0.000 }
gfCNCPoint4[25671] = {X 391.5783, Y 54.6186, Z -6.3333, A 0.000, B 0.000, C 0.000 }
gfCNCPoint4[25672] = {X 392.1572, Y 55.3496, Z -6.3333, A 0.000, B 0.000, C 0.000 }
gfCNCPoint4[25673] = {X 392.5865, Y 56.1774, Z -6.3333, A 0.000, B 0.000, C 0.000 }
gfCNCPoint4[25674] = {X 392.8506, Y 57.0718, Z -6.3333, A 0.000, B 0.000, C 0.000 }
gfCNCPoint4[25675] = {X 392.9397, Y 58.0000, Z -6.3333, A 0.000, B 0.000, C 0.000 }
gfCNCPoint4[25676] = {X 392.9395, Y 58.9744, Z -6.3333, A 0.000, B 0.000, C 0.000 }
gfCNCPoint4[25677] = {X 392.8790, Y 59.7012, Z -6.3333, A 0.000, B 0.000, C 0.000 }
gfCNCPoint4[25678] = {X 392.7108, Y 60.4109, Z -6.3333, A 0.000, B 0.000, C 0.000 }
gfCNCPoint4[25679] = {X 392.4388, Y 61.0876, Z -6.3333, A 0.000, B 0.000, C 0.000 }
gfCNCPoint4[25680] = {X 392.0555, Y 61.7360, Z -6.3333, A 0.000, B 0.000, C 0.000 }
gfCNCPoint4[25681] = {X 391.5774, Y 62.3179, Z -6.3333, A 0.000, B 0.000, C 0.000 }
gfCNCPoint4[25682] = {X 390.8820, Y 62.9185, Z -6.3333, A 0.000, B 0.000, C 0.000 }
gfCNCPoint4[25683] = {X 390.0868, Y 63.3788, Z -6.3333, A 0.000, B 0.000, C 0.000 }
gfCNCPoint4[25684] = {X 389.2196, Y 63.6827, Z -6.3333, A 0.000, B 0.000, C 0.000 }
gfCNCPoint4[25685] = {X 389.2187, Y 73.4822, Z -6.3333, A 0.000, B 0.000, C 0.000 }
gfCNCPoint4[25686] = {X 398.8187, Y 73.4832, Z -6.3333, A 0.000, B 0.000, C 0.000 }
gfCNCPoint4[25687] = {X 398.8180, Y 80.5568, Z -6.3333, A 0.000, B 0.000, C 0.000 }
gfCNCPoint4[25688] = {X 405.8026, Y 76.0836, Z -6.3333, A 0.000, B 0.000, C 0.000 }
gfCNCPoint4[25689] = {X 400.0387, Y 73.8222, Z -6.3333, A 0.000, B 0.000, C 0.000 }
gfCNCPoint4[25690] = {X 399.4375, Y 73.6211, Z -6.3333, A 0.000, B 0.000, C 0.000 }
gfCNCPoint4[25691] = {X 398.8187, Y 73.4832, Z -6.3333, A 0.000, B 0.000, C 0.000 }
gfCNCPoint4[25692] = {X 396.4187, Y 73.4829, Z -6.3333, A 0.000, B 0.000, C 0.000 }
gfCNCPoint4[25693] = {X 396.4176, Y 84.5897, Z -6.3333, A 0.000, B 0.000, C 0.000 }
gfCNCPoint4[25694] = {X 396.4175, Y 84.9441, Z -6.3333, A 0.000, B 0.000, C 0.000 }
gfCNCPoint4[25695] = {X 411.0585, Y 75.5676, Z -6.3333, A 0.000, B 0.000, C 0.000 }
gfCNCPoint4[25696] = {X 400.9168, Y 71.5886, Z -6.3333, A 0.000, B 0.000, C 0.000 }
gfCNCPoint4[25697] = {X 399.6197, Y 71.1945, Z -6.3333, A 0.000, B 0.000, C 0.000 }
gfCNCPoint4[25698] = {X 398.2765, Y 71.0108, Z -6.3333, A 0.000, B 0.000, C 0.000 }
gfCNCPoint4[25699] = {X 397.3441, Y 70.9529, Z -6.3333, A 0.000, B 0.000, C 0.000 }
gfCNCPoint4[25700] = {X 396.4189, Y 70.8232, Z -6.3333, A 0.000, B 0.000, C 0.000 }
gfCNCPoint4[25701] = {X 396.4187, Y 73.4829, Z -6.3333, A 0.000, B 0.000, C 0.000 }
gfCNCPoint4[25702] = {X 394.0187, Y 73.4827, Z -6.3333, A 0.000, B 0.000, C 0.000 }
gfCNCPoint4[25703] = {X 394.0176, Y 84.5973, Z -6.3333, A 0.000, B 0.000, C 0.000 }
gfCNCPoint4[25704] = {X 394.0181, Y 84.7624, Z -6.3333, A 0.000, B 0.000, C 0.000 }
gfCNCPoint4[25705] = {X 394.0176, Y 84.9274, Z -6.3333, A 0.000, B 0.000, C 0.000 }
gfCNCPoint4[25706] = {X 393.9672, Y 86.3330, Z -6.3333, A 0.000, B 0.000, C 0.000 }
gfCNCPoint4[25707] = {X 393.8358, Y 87.7334, Z -6.3333, A 0.000, B 0.000, C 0.000 }
gfCNCPoint4[25708] = {X 395.0761, Y 87.4777, Z -6.3333, A 0.000, B 0.000, C 0.000 }
gfCNCPoint4[25709] = {X 396.3390, Y 87.3862, Z -6.3333, A 0.000, B 0.000, C 0.000 }
gfCNCPoint4[25710] = {X 396.7288, Y 87.3713, Z -6.3333, A 0.000, B 0.000, C 0.000 }
gfCNCPoint4[25711] = {X 397.1179, Y 87.3455, Z -6.3333, A 0.000, B 0.000, C 0.000 }
gfCNCPoint4[25712] = {X 416.3144, Y 75.0516, Z -6.3333, A 0.000, B 0.000, C 0.000 }
gfCNCPoint4[25713] = {X 401.7948, Y 69.3550, Z -6.3333, A 0.000, B 0.000, C 0.000 }
gfCNCPoint4[25714] = {X 400.6812, Y 68.9849, Z -6.3333, A 0.000, B 0.000, C 0.000 }
gfCNCPoint4[25715] = {X 399.5344, Y 68.7364, Z -6.3333, A 0.000, B 0.000, C 0.000 }
gfCNCPoint4[25716] = {X 398.3675, Y 68.6122, Z -6.3333, A 0.000, B 0.000, C 0.000 }
gfCNCPoint4[25717] = {X 397.6027, Y 68.5668, Z -6.3333, A 0.000, B 0.000, C 0.000 }
gfCNCPoint4[25718] = {X 396.8439, Y 68.4611, Z -6.3333, A 0.000, B 0.000, C 0.000 }
gfCNCPoint4[25719] = {X 395.3936, Y 68.0823, Z -6.3333, A 0.000, B 0.000, C 0.000 }
gfCNCPoint4[25720] = {X 394.0193, Y 67.4842, Z -6.3333, A 0.000, B 0.000, C 0.000 }
gfCNCPoint4[25721] = {X 394.0187, Y 73.4827, Z -6.3333, A 0.000, B 0.000, C 0.000 }
gfCNCPoint4[25722] = {X 391.6187, Y 73.4825, Z -6.3333, A 0.000, B 0.000, C 0.000 }
gfCNCPoint4[25723] = {X 391.6176, Y 84.6054, Z -6.3333, A 0.000, B 0.000, C 0.000 }
gfCNCPoint4[25724] = {X 391.5816, Y 86.0255, Z -6.3333, A 0.000, B 0.000, C 0.000 }
gfCNCPoint4[25725] = {X 391.4538, Y 87.4403, Z -6.3333, A 0.000, B 0.000, C 0.000 }
gfCNCPoint4[25726] = {X 391.2295, Y 88.8722, Z -6.3333, A 0.000, B 0.000, C 0.000 }
gfCNCPoint4[25727] = {X 390.9112, Y 90.2863, Z -6.3333, A 0.000, B 0.000, C 0.000 }
gfCNCPoint4[25728] = {X 390.3349, Y 92.0501, Z -6.3333, A 0.000, B 0.000, C 0.000 }
gfCNCPoint4[25729] = {X 389.5434, Y 93.7284, Z -6.3333, A 0.000, B 0.000, C 0.000 }
gfCNCPoint4[25730] = {X 388.5491, Y 95.2951, Z -6.3333, A 0.000, B 0.000, C 0.000 }
gfCNCPoint4[25731] = {X 389.3446, Y 95.2951, Z -6.3333, A 0.000, B 0.000, C 0.000 }
gfCNCPoint4[25732] = {X 389.7639, Y 94.0857, Z -6.3333, A 0.000, B 0.000, C 0.000 }
gfCNCPoint4[25733] = {X 390.3886, Y 92.9684, Z -6.3333, A 0.000, B 0.000, C 0.000 }
gfCNCPoint4[25734] = {X 391.1993, Y 91.9778, Z -6.3333, A 0.000, B 0.000, C 0.000 }
gfCNCPoint4[25735] = {X 392.1710, Y 91.1445, Z -6.3333, A 0.000, B 0.000, C 0.000 }
gfCNCPoint4[25736] = {X 393.2736, Y 90.4943, Z -6.3333, A 0.000, B 0.000, C 0.000 }
gfCNCPoint4[25737] = {X 394.4731, Y 90.0472, Z -6.3333, A 0.000, B 0.000, C 0.000 }
gfCNCPoint4[25738] = {X 395.4148, Y 89.8537, Z -6.3333, A 0.000, B 0.000, C 0.000 }
gfCNCPoint4[25739] = {X 396.3739, Y 89.7860, Z -6.3333, A 0.000, B 0.000, C 0.000 }
gfCNCPoint4[25740] = {X 397.1502, Y 89.7499, Z -6.3333, A 0.000, B 0.000, C 0.000 }
gfCNCPoint4[25741] = {X 397.9239, Y 89.6767, Z -6.3333, A 0.000, B 0.000, C 0.000 }
gfCNCPoint4[25742] = {X 417.6088, Y 77.0726, Z -6.3333, A 0.000, B 0.000, C 0.000 }
gfCNCPoint4[25743] = {X 421.5703, Y 74.5355, Z -6.3333, A 0.000, B 0.000, C 0.000 }
gfCNCPoint4[25744] = {X 402.6729, Y 67.1214, Z -6.3333, A 0.000, B 0.000, C 0.000 }
gfCNCPoint4[25745] = {X 401.3006, Y 66.6662, Z -6.3333, A 0.000, B 0.000, C 0.000 }
gfCNCPoint4[25746] = {X 399.8872, Y 66.3623, Z -6.3333, A 0.000, B 0.000, C 0.000 }
gfCNCPoint4[25747] = {X 398.4491, Y 66.2133, Z -6.3333, A 0.000, B 0.000, C 0.000 }
gfCNCPoint4[25748] = {X 397.3049, Y 66.1054, Z -6.3333, A 0.000, B 0.000, C 0.000 }
gfCNCPoint4[25749] = {X 396.1918, Y 65.8189, Z -6.3333, A 0.000, B 0.000, C 0.000 }
gfCNCPoint4[25750] = {X 395.1377, Y 65.3607, Z -6.3333, A 0.000, B 0.000, C 0.000 }
gfCNCPoint4[25751] = {X 394.1689, Y 64.7424, Z -6.3333, A 0.000, B 0.000, C 0.000 }
gfCNCPoint4[25752] = {X 393.3095, Y 63.9793, Z -6.3333, A 0.000, B 0.000, C 0.000 }
gfCNCPoint4[25753] = {X 392.5127, Y 64.6963, Z -6.3333, A 0.000, B 0.000, C 0.000 }
gfCNCPoint4[25754] = {X 391.6195, Y 65.2890, Z -6.3333, A 0.000, B 0.000, C 0.000 }
gfCNCPoint4[25755] = {X 391.6187, Y 73.4825, Z -6.3333, A 0.000, B 0.000, C 0.000 }
gfCNCPoint4[25756] = {X 389.2187, Y 73.4822, Z -6.3333, A 0.000, B 0.000, C 0.000 }
gfCNCPoint4[25757] = {X 389.2176, Y 84.6139, Z -6.3333, A 0.000, B 0.000, C 0.000 }
gfCNCPoint4[25758] = {X 389.1557, Y 86.3199, Z -6.3333, A 0.000, B 0.000, C 0.000 }
gfCNCPoint4[25759] = {X 388.9454, Y 88.0141, Z -6.3333, A 0.000, B 0.000, C 0.000 }
gfCNCPoint4[25760] = {X 388.5881, Y 89.6835, Z -6.3333, A 0.000, B 0.000, C 0.000 }
gfCNCPoint4[25761] = {X 388.1049, Y 91.1630, Z -6.3333, A 0.000, B 0.000, C 0.000 }
gfCNCPoint4[25762] = {X 387.4410, Y 92.5709, Z -6.3333, A 0.000, B 0.000, C 0.000 }
gfCNCPoint4[25763] = {X 386.6070, Y 93.8851, Z -6.3333, A 0.000, B 0.000, C 0.000 }
gfCNCPoint4[25764] = {X 385.8749, Y 94.7997, Z -6.3333, A 0.000, B 0.000, C 0.000 }
gfCNCPoint4[25765] = {X 385.0602, Y 95.6416, Z -6.3333, A 0.000, B 0.000, C 0.000 }
gfCNCPoint4[25766] = {X 383.8004, Y 96.7249, Z -6.3333, A 0.000, B 0.000, C 0.000 }
gfCNCPoint4[25767] = {X 382.4516, Y 97.6951, Z -6.3333, A 0.000, B 0.000, C 0.000 }
gfCNCPoint4[25768] = {X 382.1884, Y 97.2937, Z -6.3333, A 0.000, B 0.000, C 0.000 }
gfCNCPoint4[25769] = {X 381.0204, Y 97.9998, Z -6.3333, A 0.000, B 0.000, C 0.000 }
gfCNCPoint4[25770] = {X 379.8039, Y 98.6188, Z -6.3333, A 0.000, B 0.000, C 0.000 }
gfCNCPoint4[25771] = {X 377.5266, Y 99.5762, Z -6.3333, A 0.000, B 0.000, C 0.000 }
gfCNCPoint4[25772] = {X 375.1867, Y 100.3684, Z -6.3333, A 0.000, B 0.000, C 0.000 }
gfCNCPoint4[25773] = {X 372.7962, Y 100.9913, Z -6.3333, A 0.000, B 0.000, C 0.000 }
gfCNCPoint4[25774] = {X 368.8820, Y 101.7461, Z -6.3333, A 0.000, B 0.000, C 0.000 }
gfCNCPoint4[25775] = {X 364.9353, Y 102.3068, Z -6.3333, A 0.000, B 0.000, C 0.000 }
gfCNCPoint4[25776] = {X 360.9658, Y 102.6723, Z -6.3333, A 0.000, B 0.000, C 0.000 }
gfCNCPoint4[25777] = {X 355.2455, Y 102.9774, Z -6.3333, A 0.000, B 0.000, C 0.000 }
gfCNCPoint4[25778] = {X 349.5185, Y 103.1074, Z -6.3333, A 0.000, B 0.000, C 0.000 }
gfCNCPoint4[25779] = {X 343.7902, Y 103.0624, Z -6.3333, A 0.000, B 0.000, C 0.000 }
gfCNCPoint4[25780] = {X 338.0660, Y 102.8424, Z -6.3333, A 0.000, B 0.000, C 0.000 }
gfCNCPoint4[25781] = {X 334.1085, Y 102.5652, Z -6.3333, A 0.000, B 0.000, C 0.000 }
gfCNCPoint4[25782] = {X 330.1660, Y 102.1230, Z -6.3333, A 0.000, B 0.000, C 0.000 }
gfCNCPoint4[25783] = {X 326.2454, Y 101.5165, Z -6.3333, A 0.000, B 0.000, C 0.000 }
gfCNCPoint4[25784] = {X 323.3900, Y 100.9107, Z -6.3333, A 0.000, B 0.000, C 0.000 }
gfCNCPoint4[25785] = {X 320.5871, Y 100.0961, Z -6.3333, A 0.000, B 0.000, C 0.000 }
gfCNCPoint4[25786] = {X 317.8518, Y 99.0773, Z -6.3333, A 0.000, B 0.000, C 0.000 }
gfCNCPoint4[25787] = {X 316.3328, Y 98.3767, Z -6.3333, A 0.000, B 0.000, C 0.000 }
gfCNCPoint4[25788] = {X 314.8778, Y 97.5515, Z -6.3333, A 0.000, B 0.000, C 0.000 }
gfCNCPoint4[25789] = {X 313.4968, Y 96.6076, Z -6.3333, A 0.000, B 0.000, C 0.000 }
gfCNCPoint4[25790] = {X 312.1996, Y 95.5516, Z -6.3333, A 0.000, B 0.000, C 0.000 }
gfCNCPoint4[25791] = {X 311.1890, Y 94.5461, Z -6.3333, A 0.000, B 0.000, C 0.000 }
gfCNCPoint4[25792] = {X 310.3048, Y 93.4280, Z -6.3333, A 0.000, B 0.000, C 0.000 }
gfCNCPoint4[25793] = {X 309.5592, Y 92.2129, Z -6.3333, A 0.000, B 0.000, C 0.000 }
gfCNCPoint4[25794] = {X 308.9630, Y 90.9180, Z -6.3333, A 0.000, B 0.000, C 0.000 }
gfCNCPoint4[25795] = {X 308.5243, Y 89.5616, Z -6.3333, A 0.000, B 0.000, C 0.000 }
gfCNCPoint4[25796] = {X 308.1796, Y 87.9321, Z -6.3333, A 0.000, B 0.000, C 0.000 }
gfCNCPoint4[25797] = {X 307.9758, Y 86.2791, Z -6.3333, A 0.000, B 0.000, C 0.000 }
gfCNCPoint4[25798] = {X 307.9147, Y 84.6146, Z -6.3333, A 0.000, B 0.000, C 0.000 }
gfCNCPoint4[25799] = {X 307.9160, Y 63.2812, Z -6.3333, A 0.000, B 0.000, C 0.000 }
gfCNCPoint4[25800] = {X 307.0567, Y 63.0559, Z -6.3333, A 0.000, B 0.000, C 0.000 }
gfCNCPoint4[25801] = {X 306.2602, Y 62.6627, Z -6.3333, A 0.000, B 0.000, C 0.000 }
gfCNCPoint4[25802] = {X 305.5589, Y 62.1176, Z -6.3333, A 0.000, B 0.000, C 0.000 }
gfCNCPoint4[25803] = {X 304.9814, Y 61.4427, Z -6.3333, A 0.000, B 0.000, C 0.000 }
gfCNCPoint4[25804] = {X 304.5512, Y 60.6655, Z -6.3333, A 0.000, B 0.000, C 0.000 }
gfCNCPoint4[25805] = {X 304.2859, Y 59.8178, Z -6.3333, A 0.000, B 0.000, C 0.000 }
gfCNCPoint4[25806] = {X 304.1962, Y 58.9341, Z -6.3333, A 0.000, B 0.000, C 0.000 }
gfCNCPoint4[25807] = {X 304.1962, Y 58.0000, Z -6.3333, A 0.000, B 0.000, C 0.000 }
gfCNCPoint4[25808] = {X 304.3065, Y 57.0209, Z -6.3333, A 0.000, B 0.000, C 0.000 }
gfCNCPoint4[25809] = {X 304.6320, Y 56.0909, Z -6.3333, A 0.000, B 0.000, C 0.000 }
gfCNCPoint4[25810] = {X 305.1562, Y 55.2566, Z -6.3333, A 0.000, B 0.000, C 0.000 }
gfCNCPoint4[25811] = {X 305.8529, Y 54.5599, Z -6.3333, A 0.000, B 0.000, C 0.000 }
gfCNCPoint4[25812] = {X 306.6871, Y 54.0357, Z -6.3333, A 0.000, B 0.000, C 0.000 }
gfCNCPoint4[25813] = {X 307.6171, Y 53.7103, Z -6.3333, A 0.000, B 0.000, C 0.000 }
gfCNCPoint4[25814] = {X 308.5962, Y 53.6000, Z -6.3333, A 0.000, B 0.000, C 0.000 }
gfCNCPoint4[25815] = {X 324.3107, Y 53.6000, Z -6.3333, A 0.000, B 0.000, C 0.000 }
gfCNCPoint4[25816] = {X 325.2898, Y 53.7103, Z -6.3333, A 0.000, B 0.000, C 0.000 }
gfCNCPoint4[25817] = {X 326.2198, Y 54.0357, Z -6.3333, A 0.000, B 0.000, C 0.000 }
gfCNCPoint4[25818] = {X 327.0540, Y 54.5599, Z -6.3333, A 0.000, B 0.000, C 0.000 }
gfCNCPoint4[25819] = {X 327.7507, Y 55.2566, Z -6.3333, A 0.000, B 0.000, C 0.000 }
gfCNCPoint4[25820] = {X 328.2750, Y 56.0909, Z -6.3333, A 0.000, B 0.000, C 0.000 }
gfCNCPoint4[25821] = {X 328.6004, Y 57.0209, Z -6.3333, A 0.000, B 0.000, C 0.000 }
gfCNCPoint4[25822] = {X 328.7107, Y 58.0000, Z -6.3333, A 0.000, B 0.000, C 0.000 }
gfCNCPoint4[25823] = {X 328.7107, Y 58.9363, Z -6.3333, A 0.000, B 0.000, C 0.000 }
gfCNCPoint4[25824] = {X 328.6171, Y 59.8190, Z -6.3333, A 0.000, B 0.000, C 0.000 }
gfCNCPoint4[25825] = {X 328.3497, Y 60.6655, Z -6.3333, A 0.000, B 0.000, C 0.000 }
gfCNCPoint4[25826] = {X 327.9192, Y 61.4418, Z -6.3333, A 0.000, B 0.000, C 0.000 }
gfCNCPoint4[25827] = {X 327.3427, Y 62.1169, Z -6.3333, A 0.000, B 0.000, C 0.000 }
gfCNCPoint4[25828] = {X 326.6434, Y 62.6638, Z -6.3333, A 0.000, B 0.000, C 0.000 }
gfCNCPoint4[25829] = {X 325.8493, Y 63.0605, Z -6.3333, A 0.000, B 0.000, C 0.000 }
gfCNCPoint4[25830] = {X 324.9921, Y 63.2912, Z -6.3333, A 0.000, B 0.000, C 0.000 }
gfCNCPoint4[25831] = {X 324.9939, Y 83.2293, Z -6.3333, A 0.000, B 0.000, C 0.000 }
gfCNCPoint4[25832] = {X 325.0074, Y 84.6143, Z -6.3333, A 0.000, B 0.000, C 0.000 }
gfCNCPoint4[25833] = {X 325.0834, Y 85.8322, Z -6.3333, A 0.000, B 0.000, C 0.000 }
gfCNCPoint4[25834] = {X 325.3003, Y 87.0331, Z -6.3333, A 0.000, B 0.000, C 0.000 }
gfCNCPoint4[25835] = {X 325.5334, Y 87.2835, Z -6.3333, A 0.000, B 0.000, C 0.000 }
gfCNCPoint4[25836] = {X 325.8189, Y 87.4719, Z -6.3333, A 0.000, B 0.000, C 0.000 }
gfCNCPoint4[25837] = {X 326.2623, Y 87.7228, Z -6.3333, A 0.000, B 0.000, C 0.000 }
gfCNCPoint4[25838] = {X 327.6908, Y 88.3151, Z -6.3333, A 0.000, B 0.000, C 0.000 }
gfCNCPoint4[25839] = {X 329.1754, Y 88.7475, Z -6.3333, A 0.000, B 0.000, C 0.000 }
gfCNCPoint4[25840] = {X 331.4458, Y 89.2202, Z -6.3333, A 0.000, B 0.000, C 0.000 }
gfCNCPoint4[25841] = {X 333.7367, Y 89.5807, Z -6.3333, A 0.000, B 0.000, C 0.000 }
gfCNCPoint4[25842] = {X 336.0424, Y 89.8283, Z -6.3333, A 0.000, B 0.000, C 0.000 }
gfCNCPoint4[25843] = {X 340.4116, Y 90.1224, Z -6.3333, A 0.000, B 0.000, C 0.000 }
gfCNCPoint4[25844] = {X 344.7880, Y 90.2762, Z -6.3333, A 0.000, B 0.000, C 0.000 }
gfCNCPoint4[25845] = {X 349.1670, Y 90.2893, Z -6.3333, A 0.000, B 0.000, C 0.000 }
gfCNCPoint4[25846] = {X 353.3143, Y 90.2210, Z -6.3333, A 0.000, B 0.000, C 0.000 }
gfCNCPoint4[25847] = {X 357.4564, Y 90.0021, Z -6.3333, A 0.000, B 0.000, C 0.000 }
gfCNCPoint4[25848] = {X 361.5878, Y 89.6331, Z -6.3333, A 0.000, B 0.000, C 0.000 }
gfCNCPoint4[25849] = {X 363.6655, Y 89.3465, Z -6.3333, A 0.000, B 0.000, C 0.000 }
gfCNCPoint4[25850] = {X 365.7242, Y 88.9451, Z -6.3333, A 0.000, B 0.000, C 0.000 }
gfCNCPoint4[25851] = {X 367.7574, Y 88.4302, Z -6.3333, A 0.000, B 0.000, C 0.000 }
gfCNCPoint4[25852] = {X 368.6800, Y 88.1199, Z -6.3333, A 0.000, B 0.000, C 0.000 }
gfCNCPoint4[25853] = {X 369.5620, Y 87.7082, Z -6.3333, A 0.000, B 0.000, C 0.000 }
gfCNCPoint4[25854] = {X 370.3923, Y 87.2002, Z -6.3333, A 0.000, B 0.000, C 0.000 }
gfCNCPoint4[25855] = {X 370.5199, Y 87.0674, Z -6.3333, A 0.000, B 0.000, C 0.000 }
gfCNCPoint4[25856] = {X 370.5856, Y 86.8955, Z -6.3333, A 0.000, B 0.000, C 0.000 }
gfCNCPoint4[25857] = {X 370.7759, Y 85.3673, Z -6.3333, A 0.000, B 0.000, C 0.000 }
gfCNCPoint4[25858] = {X 370.8394, Y 83.8287, Z -6.3333, A 0.000, B 0.000, C 0.000 }
gfCNCPoint4[25859] = {X 370.8381, Y 63.2810, Z -6.3333, A 0.000, B 0.000, C 0.000 }
gfCNCPoint4[25860] = {X 369.9791, Y 63.0557, Z -6.3333, A 0.000, B 0.000, C 0.000 }
gfCNCPoint4[25861] = {X 369.1827, Y 62.6624, Z -6.3333, A 0.000, B 0.000, C 0.000 }
gfCNCPoint4[25862] = {X 368.4816, Y 62.1172, Z -6.3333, A 0.000, B 0.000, C 0.000 }
gfCNCPoint4[25863] = {X 367.9042, Y 61.4423, Z -6.3333, A 0.000, B 0.000, C 0.000 }
gfCNCPoint4[25864] = {X 367.4742, Y 60.6653, Z -6.3333, A 0.000, B 0.000, C 0.000 }
gfCNCPoint4[25865] = {X 367.2089, Y 59.8177, Z -6.3333, A 0.000, B 0.000, C 0.000 }
gfCNCPoint4[25866] = {X 367.1193, Y 58.9341, Z -6.3333, A 0.000, B 0.000, C 0.000 }
gfCNCPoint4[25867] = {X 367.1193, Y 58.0000, Z -6.3333, A 0.000, B 0.000, C 0.000 }
gfCNCPoint4[25868] = {X 367.2296, Y 57.0209, Z -6.3333, A 0.000, B 0.000, C 0.000 }
gfCNCPoint4[25869] = {X 367.5550, Y 56.0909, Z -6.3333, A 0.000, B 0.000, C 0.000 }
gfCNCPoint4[25870] = {X 368.0792, Y 55.2566, Z -6.3333, A 0.000, B 0.000, C 0.000 }
gfCNCPoint4[25871] = {X 368.7759, Y 54.5599, Z -6.3333, A 0.000, B 0.000, C 0.000 }
gfCNCPoint4[25872] = {X 369.6102, Y 54.0357, Z -6.3333, A 0.000, B 0.000, C 0.000 }
gfCNCPoint4[25873] = {X 370.5402, Y 53.7103, Z -6.3333, A 0.000, B 0.000, C 0.000 }
gfCNCPoint4[25874] = {X 371.5193, Y 53.6000, Z -6.3333, A 0.000, B 0.000, C 0.000 }
gfCNCPoint4[25875] = {X 388.0597, Y 53.6000, Z -6.3333, A 0.000, B 0.000, C 0.000 }
gfCNCPoint4[25876] = {X 389.0388, Y 53.7103, Z -6.3333, A 0.000, B 0.000, C 0.000 }
gfCNCPoint4[25877] = {X 389.9688, Y 54.0357, Z -6.3333, A 0.000, B 0.000, C 0.000 }
gfCNCPoint4[25878] = {X 390.8030, Y 54.5599, Z -6.3333, A 0.000, B 0.000, C 0.000 }
gfCNCPoint4[25879] = {X 391.4997, Y 55.2566, Z -6.3333, A 0.000, B 0.000, C 0.000 }
gfCNCPoint4[25880] = {X 392.0239, Y 56.0909, Z -6.3333, A 0.000, B 0.000, C 0.000 }
gfCNCPoint4[25881] = {X 392.3494, Y 57.0209, Z -6.3333, A 0.000, B 0.000, C 0.000 }
gfCNCPoint4[25882] = {X 392.4597, Y 58.0000, Z -6.3333, A 0.000, B 0.000, C 0.000 }
gfCNCPoint4[25883] = {X 392.4595, Y 58.9704, Z -6.3333, A 0.000, B 0.000, C 0.000 }
gfCNCPoint4[25884] = {X 392.3411, Y 59.9485, Z -6.3333, A 0.000, B 0.000, C 0.000 }
gfCNCPoint4[25885] = {X 392.0081, Y 60.8758, Z -6.3333, A 0.000, B 0.000, C 0.000 }
gfCNCPoint4[25886] = {X 391.5655, Y 61.5936, Z -6.3333, A 0.000, B 0.000, C 0.000 }
gfCNCPoint4[25887] = {X 390.9948, Y 62.2143, Z -6.3333, A 0.000, B 0.000, C 0.000 }
gfCNCPoint4[25888] = {X 390.3166, Y 62.7154, Z -6.3333, A 0.000, B 0.000, C 0.000 }
gfCNCPoint4[25889] = {X 389.5557, Y 63.0788, Z -6.3333, A 0.000, B 0.000, C 0.000 }
gfCNCPoint4[25890] = {X 388.7396, Y 63.2911, Z -6.3333, A 0.000, B 0.000, C 0.000 }
gfCNCPoint4[25891] = {X 388.7396, Y 83.9247, Z -6.3333, A 0.000, B 0.000, C 0.000 }
gfCNCPoint4[25892] = {X 388.7376, Y 84.6149, Z -6.3333, A 0.000, B 0.000, C 0.000 }
gfCNCPoint4[25893] = {X 388.6774, Y 86.2800, Z -6.3333, A 0.000, B 0.000, C 0.000 }
gfCNCPoint4[25894] = {X 388.4722, Y 87.9334, Z -6.3333, A 0.000, B 0.000, C 0.000 }
gfCNCPoint4[25895] = {X 388.1236, Y 89.5626, Z -6.3333, A 0.000, B 0.000, C 0.000 }
gfCNCPoint4[25896] = {X 387.5877, Y 91.1607, Z -6.3333, A 0.000, B 0.000, C 0.000 }
gfCNCPoint4[25897] = {X 386.8330, Y 92.6678, Z -6.3333, A 0.000, B 0.000, C 0.000 }
gfCNCPoint4[25898] = {X 385.8745, Y 94.0542, Z -6.3333, A 0.000, B 0.000, C 0.000 }
gfCNCPoint4[25899] = {X 384.7309, Y 95.2924, Z -6.3333, A 0.000, B 0.000, C 0.000 }
gfCNCPoint4[25900] = {X 383.5030, Y 96.3481, Z -6.3333, A 0.000, B 0.000, C 0.000 }
gfCNCPoint4[25901] = {X 382.1884, Y 97.2937, Z -6.3333, A 0.000, B 0.000, C 0.000 }
gfCNCPoint4[25902] = {X 382.4516, Y 97.6951, Z -6.3333, A 0.000, B 0.000, C 0.000 }
gfCNCPoint4[25903] = {X 391.5259, Y 97.6951, Z -6.3333, A 0.000, B 0.000, C 0.000 }
gfCNCPoint4[25904] = {X 391.5259, Y 97.0659, Z -6.3333, A 0.000, B 0.000, C 0.000 }
gfCNCPoint4[25905] = {X 391.6197, Y 96.1142, Z -6.3333, A 0.000, B 0.000, C 0.000 }
gfCNCPoint4[25906] = {X 391.8972, Y 95.1990, Z -6.3333, A 0.000, B 0.000, C 0.000 }
gfCNCPoint4[25907] = {X 392.3478, Y 94.3556, Z -6.3333, A 0.000, B 0.000, C 0.000 }
gfCNCPoint4[25908] = {X 392.9544, Y 93.6162, Z -6.3333, A 0.000, B 0.000, C 0.000 }
gfCNCPoint4[25909] = {X 393.6934, Y 93.0093, Z -6.3333, A 0.000, B 0.000, C 0.000 }
gfCNCPoint4[25910] = {X 394.5367, Y 92.5581, Z -6.3333, A 0.000, B 0.000, C 0.000 }
gfCNCPoint4[25911] = {X 395.4517, Y 92.2801, Z -6.3333, A 0.000, B 0.000, C 0.000 }
gfCNCPoint4[25912] = {X 396.4034, Y 92.1859, Z -6.3333, A 0.000, B 0.000, C 0.000 }
gfCNCPoint4[25913] = {X 397.3158, Y 92.1442, Z -6.3333, A 0.000, B 0.000, C 0.000 }
gfCNCPoint4[25914] = {X 398.2251, Y 92.0578, Z -6.3333, A 0.000, B 0.000, C 0.000 }
gfCNCPoint4[25915] = {X 398.7531, Y 91.9294, Z -6.3333, A 0.000, B 0.000, C 0.000 }
gfCNCPoint4[25916] = {X 399.2394, Y 91.6869, Z -6.3333, A 0.000, B 0.000, C 0.000 }
gfCNCPoint4[25917] = {X 426.8262, Y 74.0195, Z -6.3333, A 0.000, B 0.000, C 0.000 }
gfCNCPoint4[25918] = {X 403.5509, Y 64.8878, Z -6.3333, A 0.000, B 0.000, C 0.000 }
gfCNCPoint4[25919] = {X 401.9166, Y 64.3466, Z -6.3333, A 0.000, B 0.000, C 0.000 }
gfCNCPoint4[25920] = {X 400.2330, Y 63.9872, Z -6.3333, A 0.000, B 0.000, C 0.000 }
gfCNCPoint4[25921] = {X 398.5201, Y 63.8139, Z -6.3333, A 0.000, B 0.000, C 0.000 }
gfCNCPoint4[25922] = {X 397.5545, Y 63.7098, Z -6.3333, A 0.000, B 0.000, C 0.000 }
gfCNCPoint4[25923] = {X 396.6286, Y 63.4166, Z -6.3333, A 0.000, B 0.000, C 0.000 }
gfCNCPoint4[25924] = {X 395.7791, Y 62.9457, Z -6.3333, A 0.000, B 0.000, C 0.000 }
gfCNCPoint4[25925] = {X 395.0397, Y 62.3160, Z -6.3333, A 0.000, B 0.000, C 0.000 }
gfCNCPoint4[25926] = {X 394.4660, Y 61.5934, Z -6.3333, A 0.000, B 0.000, C 0.000 }
gfCNCPoint4[25927] = {X 394.0386, Y 60.7757, Z -6.3333, A 0.000, B 0.000, C 0.000 }
gfCNCPoint4[25928] = {X 393.7727, Y 59.8921, Z -6.3333, A 0.000, B 0.000, C 0.000 }
gfCNCPoint4[25929] = {X 393.6779, Y 58.9744, Z -6.3333, A 0.000, B 0.000, C 0.000 }
gfCNCPoint4[25930] = {X 393.6777, Y 58.0000, Z -6.3333, A 0.000, B 0.000, C 0.000 }
gfCNCPoint4[25931] = {X 393.7668, Y 57.0718, Z -6.3333, A 0.000, B 0.000, C 0.000 }
gfCNCPoint4[25932] = {X 394.0309, Y 56.1774, Z -6.3333, A 0.000, B 0.000, C 0.000 }
gfCNCPoint4[25933] = {X 394.4602, Y 55.3496, Z -6.3333, A 0.000, B 0.000, C 0.000 }
gfCNCPoint4[25934] = {X 395.0391, Y 54.6186, Z -6.3333, A 0.000, B 0.000, C 0.000 }
gfCNCPoint4[25935] = {X 395.7864, Y 53.9833, Z -6.3333, A 0.000, B 0.000, C 0.000 }
gfCNCPoint4[25936] = {X 396.6455, Y 53.5102, Z -6.3333, A 0.000, B 0.000, C 0.000 }
gfCNCPoint4[25937] = {X 397.5819, Y 53.2186, Z -6.3333, A 0.000, B 0.000, C 0.000 }
gfCNCPoint4[25938] = {X 398.5577, Y 53.1200, Z -6.3333, A 0.000, B 0.000, C 0.000 }
gfCNCPoint4[25939] = {X 419.4886, Y 53.1200, Z -6.3333, A 0.000, B 0.000, C 0.000 }
gfCNCPoint4[25940] = {X 420.5533, Y 53.2376, Z -6.3333, A 0.000, B 0.000, C 0.000 }
gfCNCPoint4[25941] = {X 421.5667, Y 53.5846, Z -6.3333, A 0.000, B 0.000, C 0.000 }
gfCNCPoint4[25942] = {X 422.4800, Y 54.1444, Z -6.3333, A 0.000, B 0.000, C 0.000 }
gfCNCPoint4[25943] = {X 423.2492, Y 54.8899, Z -6.3333, A 0.000, B 0.000, C 0.000 }
gfCNCPoint4[25944] = {X 423.8371, Y 55.7854, Z -6.3333, A 0.000, B 0.000, C 0.000 }
gfCNCPoint4[25945] = {X 424.2156, Y 56.7875, Z -6.3333, A 0.000, B 0.000, C 0.000 }
gfCNCPoint4[25946] = {X 424.3662, Y 57.8480, Z -6.3333, A 0.000, B 0.000, C 0.000 }
gfCNCPoint4[25947] = {X 429.8190, Y 59.9725, Z -6.3333, A 0.000, B 0.000, C 0.000 }
gfCNCPoint4[25948] = {X 457.2982, Y 70.8754, Z -6.3333, A 0.000, B 0.000, C 0.000 }
gfCNCPoint4[25949] = {X 457.2985, Y 63.6739, Z -6.3333, A 0.000, B 0.000, C 0.000 }
gfCNCPoint4[25950] = {X 456.2905, Y 63.3055, Z -6.3333, A 0.000, B 0.000, C 0.000 }
gfCNCPoint4[25951] = {X 455.3873, Y 62.7256, Z -6.3333, A 0.000, B 0.000, C 0.000 }
gfCNCPoint4[25952] = {X 454.6328, Y 61.9622, Z -6.3333, A 0.000, B 0.000, C 0.000 }
gfCNCPoint4[25953] = {X 454.0634, Y 61.0524, Z -6.3333, A 0.000, B 0.000, C 0.000 }
gfCNCPoint4[25954] = {X 453.7066, Y 60.0401, Z -6.3333, A 0.000, B 0.000, C 0.000 }
gfCNCPoint4[25955] = {X 453.5798, Y 58.9744, Z -6.3333, A 0.000, B 0.000, C 0.000 }
gfCNCPoint4[25956] = {X 453.5796, Y 58.0000, Z -6.3333, A 0.000, B 0.000, C 0.000 }
gfCNCPoint4[25957] = {X 453.6734, Y 57.0480, Z -6.3333, A 0.000, B 0.000, C 0.000 }
gfCNCPoint4[25958] = {X 453.9511, Y 56.1325, Z -6.3333, A 0.000, B 0.000, C 0.000 }
gfCNCPoint4[25959] = {X 454.4020, Y 55.2888, Z -6.3333, A 0.000, B 0.000, C 0.000 }
gfCNCPoint4[25960] = {X 455.0089, Y 54.5493, Z -6.3333, A 0.000, B 0.000, C 0.000 }
gfCNCPoint4[25961] = {X 455.7484, Y 53.9424, Z -6.3333, A 0.000, B 0.000, C 0.000 }
gfCNCPoint4[25962] = {X 456.5921, Y 53.4915, Z -6.3333, A 0.000, B 0.000, C 0.000 }
gfCNCPoint4[25963] = {X 457.5076, Y 53.2138, Z -6.3333, A 0.000, B 0.000, C 0.000 }
gfCNCPoint4[25964] = {X 458.4596, Y 53.1200, Z -6.3333, A 0.000, B 0.000, C 0.000 }
gfCNCPoint4[25965] = {X 475.0000, Y 53.1200, Z -6.3333, A 0.000, B 0.000, C 0.000 }
gfCNCPoint4[25966] = {X 475.9520, Y 53.2138, Z -6.3333, A 0.000, B 0.000, C 0.000 }
gfCNCPoint4[25967] = {X 476.8675, Y 53.4915, Z -6.3333, A 0.000, B 0.000, C 0.000 }
gfCNCPoint4[25968] = {X 477.7112, Y 53.9424, Z -6.3333, A 0.000, B 0.000, C 0.000 }
gfCNCPoint4[25969] = {X 478.4507, Y 54.5493, Z -6.3333, A 0.000, B 0.000, C 0.000 }
gfCNCPoint4[25970] = {X 479.0576, Y 55.2888, Z -6.3333, A 0.000, B 0.000, C 0.000 }
gfCNCPoint4[25971] = {X 479.5085, Y 56.1325, Z -6.3333, A 0.000, B 0.000, C 0.000 }
gfCNCPoint4[25972] = {X 479.7862, Y 57.0480, Z -6.3333, A 0.000, B 0.000, C 0.000 }
gfCNCPoint4[25973] = {X 479.8800, Y 58.0000, Z -6.3333, A 0.000, B 0.000, C 0.000 }
gfCNCPoint4[25974] = {X 479.8798, Y 58.9744, Z -6.3333, A 0.000, B 0.000, C 0.000 }
gfCNCPoint4[25975] = {X 479.7530, Y 60.0402, Z -6.3333, A 0.000, B 0.000, C 0.000 }
gfCNCPoint4[25976] = {X 479.3962, Y 61.0525, Z -6.3333, A 0.000, B 0.000, C 0.000 }
gfCNCPoint4[25977] = {X 478.8267, Y 61.9624, Z -6.3333, A 0.000, B 0.000, C 0.000 }
gfCNCPoint4[25978] = {X 478.0721, Y 62.7257, Z -6.3333, A 0.000, B 0.000, C 0.000 }
gfCNCPoint4[25979] = {X 477.1689, Y 63.3056, Z -6.3333, A 0.000, B 0.000, C 0.000 }
gfCNCPoint4[25980] = {X 476.1607, Y 63.6740, Z -6.3333, A 0.000, B 0.000, C 0.000 }
gfCNCPoint4[25981] = {X 476.1612, Y 92.3309, Z -6.3333, A 0.000, B 0.000, C 0.000 }
gfCNCPoint4[25982] = {X 476.3596, Y 92.3890, Z -6.3333, A 0.000, B 0.000, C 0.000 }
gfCNCPoint4[25983] = {X 476.5565, Y 92.4519, Z -6.3333, A 0.000, B 0.000, C 0.000 }
gfCNCPoint4[25984] = {X 477.4763, Y 92.8688, Z -6.3333, A 0.000, B 0.000, C 0.000 }
gfCNCPoint4[25985] = {X 478.2900, Y 93.4669, Z -6.3333, A 0.000, B 0.000, C 0.000 }
gfCNCPoint4[25986] = {X 478.9625, Y 94.2202, Z -6.3333, A 0.000, B 0.000, C 0.000 }
gfCNCPoint4[25987] = {X 479.4648, Y 95.0963, Z -6.3333, A 0.000, B 0.000, C 0.000 }
gfCNCPoint4[25988] = {X 479.7751, Y 96.0573, Z -6.3333, A 0.000, B 0.000, C 0.000 }
gfCNCPoint4[25989] = {X 479.8800, Y 97.0617, Z -6.3333, A 0.000, B 0.000, C 0.000 }
gfCNCPoint4[25990] = {X 479.8800, Y 97.6951, Z -6.3333, A 0.000, B 0.000, C 0.000 }
gfCNCPoint4[25991] = {X 479.4000, Y 97.6951, Z -6.3333, A 0.000, B 0.000, C 0.000 }
gfCNCPoint4[25992] = {X 479.4000, Y 98.0000, Z -6.3333, A 0.000, B 0.000, C 0.000 }
gfCNCPoint4[25993] = {X 479.2897, Y 98.9791, Z -6.3333, A 0.000, B 0.000, C 0.000 }
gfCNCPoint4[25994] = {X 478.9643, Y 99.9091, Z -6.3333, A 0.000, B 0.000, C 0.000 }
gfCNCPoint4[25995] = {X 478.4401, Y 100.7434, Z -6.3333, A 0.000, B 0.000, C 0.000 }
gfCNCPoint4[25996] = {X 477.7434, Y 101.4401, Z -6.3333, A 0.000, B 0.000, C 0.000 }
gfCNCPoint4[25997] = {X 476.9091, Y 101.9643, Z -6.3333, A 0.000, B 0.000, C 0.000 }
gfCNCPoint4[25998] = {X 475.9791, Y 102.2897, Z -6.3333, A 0.000, B 0.000, C 0.000 }
gfCNCPoint4[25999] = {X 475.0000, Y 102.4000, Z -6.3333, A 0.000, B 0.000, C 0.000 }
gfCNCPoint4[26000] = {X 458.4596, Y 102.4000, Z -6.3333, A 0.000, B 0.000, C 0.000 }
gfCNCPoint4[26001] = {X 457.4805, Y 102.2897, Z -6.3333, A 0.000, B 0.000, C 0.000 }
gfCNCPoint4[26002] = {X 456.5505, Y 101.9643, Z -6.3333, A 0.000, B 0.000, C 0.000 }
gfCNCPoint4[26003] = {X 455.7162, Y 101.4401, Z -6.3333, A 0.000, B 0.000, C 0.000 }
gfCNCPoint4[26004] = {X 455.0195, Y 100.7434, Z -6.3333, A 0.000, B 0.000, C 0.000 }
gfCNCPoint4[26005] = {X 454.4953, Y 99.9091, Z -6.3333, A 0.000, B 0.000, C 0.000 }
gfCNCPoint4[26006] = {X 454.1699, Y 98.9791, Z -6.3333, A 0.000, B 0.000, C 0.000 }
gfCNCPoint4[26007] = {X 454.0596, Y 98.0000, Z -6.3333, A 0.000, B 0.000, C 0.000 }
gfCNCPoint4[26008] = {X 454.0596, Y 97.0659, Z -6.3333, A 0.000, B 0.000, C 0.000 }
gfCNCPoint4[26009] = {X 454.1492, Y 96.1826, Z -6.3333, A 0.000, B 0.000, C 0.000 }
gfCNCPoint4[26010] = {X 454.4143, Y 95.3353, Z -6.3333, A 0.000, B 0.000, C 0.000 }
gfCNCPoint4[26011] = {X 454.8440, Y 94.5584, Z -6.3333, A 0.000, B 0.000, C 0.000 }
gfCNCPoint4[26012] = {X 455.4210, Y 93.8836, Z -6.3333, A 0.000, B 0.000, C 0.000 }
gfCNCPoint4[26013] = {X 456.1217, Y 93.3384, Z -6.3333, A 0.000, B 0.000, C 0.000 }
gfCNCPoint4[26014] = {X 456.9176, Y 92.9450, Z -6.3333, A 0.000, B 0.000, C 0.000 }
gfCNCPoint4[26015] = {X 457.7763, Y 92.7193, Z -6.3333, A 0.000, B 0.000, C 0.000 }
gfCNCPoint4[26016] = {X 457.7763, Y 85.6495, Z -6.3333, A 0.000, B 0.000, C 0.000 }
gfCNCPoint4[26017] = {X 444.8689, Y 80.5898, Z -6.3333, A 0.000, B 0.000, C 0.000 }
gfCNCPoint4[26018] = {X 420.1042, Y 96.6317, Z -6.3333, A 0.000, B 0.000, C 0.000 }
gfCNCPoint4[26019] = {X 420.1067, Y 97.0659, Z -6.3333, A 0.000, B 0.000, C 0.000 }
gfCNCPoint4[26020] = {X 420.1067, Y 98.0000, Z -6.3333, A 0.000, B 0.000, C 0.000 }
gfCNCPoint4[26021] = {X 419.9964, Y 98.9791, Z -6.3333, A 0.000, B 0.000, C 0.000 }
gfCNCPoint4[26022] = {X 419.6710, Y 99.9091, Z -6.3333, A 0.000, B 0.000, C 0.000 }
gfCNCPoint4[26023] = {X 419.1468, Y 100.7434, Z -6.3333, A 0.000, B 0.000, C 0.000 }
gfCNCPoint4[26024] = {X 418.4501, Y 101.4401, Z -6.3333, A 0.000, B 0.000, C 0.000 }
gfCNCPoint4[26025] = {X 417.6158, Y 101.9643, Z -6.3333, A 0.000, B 0.000, C 0.000 }
gfCNCPoint4[26026] = {X 416.6858, Y 102.2897, Z -6.3333, A 0.000, B 0.000, C 0.000 }
gfCNCPoint4[26027] = {X 415.7067, Y 102.4000, Z -6.3333, A 0.000, B 0.000, C 0.000 }
gfCNCPoint4[26028] = {X 396.4059, Y 102.4000, Z -6.3333, A 0.000, B 0.000, C 0.000 }
gfCNCPoint4[26029] = {X 395.4269, Y 102.2897, Z -6.3333, A 0.000, B 0.000, C 0.000 }
gfCNCPoint4[26030] = {X 394.4969, Y 101.9643, Z -6.3333, A 0.000, B 0.000, C 0.000 }
gfCNCPoint4[26031] = {X 393.6626, Y 101.4401, Z -6.3333, A 0.000, B 0.000, C 0.000 }
gfCNCPoint4[26032] = {X 392.9659, Y 100.7434, Z -6.3333, A 0.000, B 0.000, C 0.000 }
gfCNCPoint4[26033] = {X 392.4417, Y 99.9091, Z -6.3333, A 0.000, B 0.000, C 0.000 }
gfCNCPoint4[26034] = {X 392.1163, Y 98.9791, Z -6.3333, A 0.000, B 0.000, C 0.000 }
gfCNCPoint4[26035] = {X 392.0059, Y 98.0000, Z -6.3333, A 0.000, B 0.000, C 0.000 }
gfCNCPoint4[26036] = {X 392.0059, Y 97.0659, Z -6.3333, A 0.000, B 0.000, C 0.000 }
gfCNCPoint4[26037] = {X 392.1163, Y 96.0865, Z -6.3333, A 0.000, B 0.000, C 0.000 }
gfCNCPoint4[26038] = {X 392.4420, Y 95.1562, Z -6.3333, A 0.000, B 0.000, C 0.000 }
gfCNCPoint4[26039] = {X 392.9666, Y 94.3217, Z -6.3333, A 0.000, B 0.000, C 0.000 }
gfCNCPoint4[26040] = {X 393.6637, Y 93.6250, Z -6.3333, A 0.000, B 0.000, C 0.000 }
gfCNCPoint4[26041] = {X 394.4985, Y 93.1009, Z -6.3333, A 0.000, B 0.000, C 0.000 }
gfCNCPoint4[26042] = {X 395.4290, Y 92.7758, Z -6.3333, A 0.000, B 0.000, C 0.000 }
gfCNCPoint4[26043] = {X 396.4085, Y 92.6659, Z -6.3333, A 0.000, B 0.000, C 0.000 }
gfCNCPoint4[26044] = {X 397.3478, Y 92.6231, Z -6.3333, A 0.000, B 0.000, C 0.000 }
gfCNCPoint4[26045] = {X 398.2838, Y 92.5342, Z -6.3333, A 0.000, B 0.000, C 0.000 }
gfCNCPoint4[26046] = {X 398.9171, Y 92.3805, Z -6.3333, A 0.000, B 0.000, C 0.000 }
gfCNCPoint4[26047] = {X 399.5003, Y 92.0898, Z -6.3333, A 0.000, B 0.000, C 0.000 }
gfCNCPoint4[26048] = {X 405.0421, Y 88.5194, Z -6.3333, A 0.000, B 0.000, C 0.000 }
gfCNCPoint4[26049] = {X 427.8781, Y 73.9166, Z -6.3333, A 0.000, B 0.000, C 0.000 }
gfCNCPoint4[26050] = {X 403.7263, Y 64.4410, Z -6.3333, A 0.000, B 0.000, C 0.000 }
gfCNCPoint4[26051] = {X 402.0391, Y 63.8825, Z -6.3333, A 0.000, B 0.000, C 0.000 }
gfCNCPoint4[26052] = {X 400.3010, Y 63.5120, Z -6.3333, A 0.000, B 0.000, C 0.000 }
gfCNCPoint4[26053] = {X 398.5327, Y 63.3340, Z -6.3333, A 0.000, B 0.000, C 0.000 }
gfCNCPoint4[26054] = {X 397.5577, Y 63.2189, Z -6.3333, A 0.000, B 0.000, C 0.000 }
gfCNCPoint4[26055] = {X 396.6326, Y 62.8905, Z -6.3333, A 0.000, B 0.000, C 0.000 }
gfCNCPoint4[26056] = {X 395.8032, Y 62.3652, Z -6.3333, A 0.000, B 0.000, C 0.000 }
gfCNCPoint4[26057] = {X 395.1110, Y 61.6690, Z -6.3333, A 0.000, B 0.000, C 0.000 }
gfCNCPoint4[26058] = {X 394.5904, Y 60.8367, Z -6.3333, A 0.000, B 0.000, C 0.000 }
gfCNCPoint4[26059] = {X 394.2672, Y 59.9097, Z -6.3333, A 0.000, B 0.000, C 0.000 }
gfCNCPoint4[26060] = {X 394.1577, Y 58.9341, Z -6.3333, A 0.000, B 0.000, C 0.000 }
gfCNCPoint4[26061] = {X 394.1577, Y 58.0000, Z -6.3333, A 0.000, B 0.000, C 0.000 }
gfCNCPoint4[26062] = {X 394.2680, Y 57.0209, Z -6.3333, A 0.000, B 0.000, C 0.000 }
gfCNCPoint4[26063] = {X 394.5935, Y 56.0909, Z -6.3333, A 0.000, B 0.000, C 0.000 }
gfCNCPoint4[26064] = {X 395.1177, Y 55.2566, Z -6.3333, A 0.000, B 0.000, C 0.000 }
gfCNCPoint4[26065] = {X 395.8144, Y 54.5599, Z -6.3333, A 0.000, B 0.000, C 0.000 }
gfCNCPoint4[26066] = {X 396.6486, Y 54.0357, Z -6.3333, A 0.000, B 0.000, C 0.000 }
gfCNCPoint4[26067] = {X 397.5786, Y 53.7103, Z -6.3333, A 0.000, B 0.000, C 0.000 }
gfCNCPoint4[26068] = {X 398.5577, Y 53.6000, Z -6.3333, A 0.000, B 0.000, C 0.000 }
gfCNCPoint4[26069] = {X 419.4886, Y 53.6000, Z -6.3333, A 0.000, B 0.000, C 0.000 }
gfCNCPoint4[26070] = {X 420.4677, Y 53.7103, Z -6.3333, A 0.000, B 0.000, C 0.000 }
gfCNCPoint4[26071] = {X 421.3977, Y 54.0357, Z -6.3333, A 0.000, B 0.000, C 0.000 }
gfCNCPoint4[26072] = {X 422.2320, Y 54.5599, Z -6.3333, A 0.000, B 0.000, C 0.000 }
gfCNCPoint4[26073] = {X 422.9287, Y 55.2566, Z -6.3333, A 0.000, B 0.000, C 0.000 }
gfCNCPoint4[26074] = {X 423.4529, Y 56.0909, Z -6.3333, A 0.000, B 0.000, C 0.000 }
gfCNCPoint4[26075] = {X 423.7783, Y 57.0209, Z -6.3333, A 0.000, B 0.000, C 0.000 }
gfCNCPoint4[26076] = {X 423.8886, Y 58.0000, Z -6.3333, A 0.000, B 0.000, C 0.000 }
gfCNCPoint4[26077] = {X 423.8886, Y 58.1771, Z -6.3333, A 0.000, B 0.000, C 0.000 }
gfCNCPoint4[26078] = {X 429.6420, Y 60.4187, Z -6.3333, A 0.000, B 0.000, C 0.000 }
gfCNCPoint4[26079] = {X 457.7782, Y 71.5822, Z -6.3333, A 0.000, B 0.000, C 0.000 }
gfCNCPoint4[26080] = {X 457.7785, Y 63.2810, Z -6.3333, A 0.000, B 0.000, C 0.000 }
gfCNCPoint4[26081] = {X 456.9195, Y 63.0557, Z -6.3333, A 0.000, B 0.000, C 0.000 }
gfCNCPoint4[26082] = {X 456.1231, Y 62.6624, Z -6.3333, A 0.000, B 0.000, C 0.000 }
gfCNCPoint4[26083] = {X 455.4220, Y 62.1173, Z -6.3333, A 0.000, B 0.000, C 0.000 }
gfCNCPoint4[26084] = {X 454.8446, Y 61.4424, Z -6.3333, A 0.000, B 0.000, C 0.000 }
gfCNCPoint4[26085] = {X 454.4145, Y 60.6653, Z -6.3333, A 0.000, B 0.000, C 0.000 }
gfCNCPoint4[26086] = {X 454.1492, Y 59.8177, Z -6.3333, A 0.000, B 0.000, C 0.000 }
gfCNCPoint4[26087] = {X 454.0596, Y 58.9341, Z -6.3333, A 0.000, B 0.000, C 0.000 }
gfCNCPoint4[26088] = {X 454.0596, Y 58.0000, Z -6.3333, A 0.000, B 0.000, C 0.000 }
gfCNCPoint4[26089] = {X 454.1699, Y 57.0209, Z -6.3333, A 0.000, B 0.000, C 0.000 }
gfCNCPoint4[26090] = {X 454.4953, Y 56.0909, Z -6.3333, A 0.000, B 0.000, C 0.000 }
gfCNCPoint4[26091] = {X 455.0195, Y 55.2566, Z -6.3333, A 0.000, B 0.000, C 0.000 }
gfCNCPoint4[26092] = {X 455.7162, Y 54.5599, Z -6.3333, A 0.000, B 0.000, C 0.000 }
gfCNCPoint4[26093] = {X 456.5505, Y 54.0357, Z -6.3333, A 0.000, B 0.000, C 0.000 }
gfCNCPoint4[26094] = {X 457.4805, Y 53.7103, Z -6.3333, A 0.000, B 0.000, C 0.000 }
gfCNCPoint4[26095] = {X 458.4596, Y 53.6000, Z -6.3333, A 0.000, B 0.000, C 0.000 }
gfCNCPoint4[26096] = {X 475.0000, Y 53.6000, Z -6.3333, A 0.000, B 0.000, C 0.000 }
gfCNCPoint4[26097] = {X 475.9791, Y 53.7103, Z -6.3333, A 0.000, B 0.000, C 0.000 }
gfCNCPoint4[26098] = {X 476.9091, Y 54.0357, Z -6.3333, A 0.000, B 0.000, C 0.000 }
gfCNCPoint4[26099] = {X 477.7434, Y 54.5599, Z -6.3333, A 0.000, B 0.000, C 0.000 }
gfCNCPoint4[26100] = {X 478.4401, Y 55.2566, Z -6.3333, A 0.000, B 0.000, C 0.000 }
gfCNCPoint4[26101] = {X 478.9643, Y 56.0909, Z -6.3333, A 0.000, B 0.000, C 0.000 }
gfCNCPoint4[26102] = {X 479.2897, Y 57.0209, Z -6.3333, A 0.000, B 0.000, C 0.000 }
gfCNCPoint4[26103] = {X 479.4000, Y 58.0000, Z -6.3333, A 0.000, B 0.000, C 0.000 }
gfCNCPoint4[26104] = {X 479.3998, Y 58.9704, Z -6.3333, A 0.000, B 0.000, C 0.000 }
gfCNCPoint4[26105] = {X 479.3040, Y 59.8482, Z -6.3333, A 0.000, B 0.000, C 0.000 }
gfCNCPoint4[26106] = {X 479.0348, Y 60.6892, Z -6.3333, A 0.000, B 0.000, C 0.000 }
gfCNCPoint4[26107] = {X 478.6031, Y 61.4595, Z -6.3333, A 0.000, B 0.000, C 0.000 }
gfCNCPoint4[26108] = {X 478.0262, Y 62.1281, Z -6.3333, A 0.000, B 0.000, C 0.000 }
gfCNCPoint4[26109] = {X 477.3275, Y 62.6681, Z -6.3333, A 0.000, B 0.000, C 0.000 }
gfCNCPoint4[26110] = {X 476.5350, Y 63.0576, Z -6.3333, A 0.000, B 0.000, C 0.000 }
gfCNCPoint4[26111] = {X 475.6807, Y 63.2811, Z -6.3333, A 0.000, B 0.000, C 0.000 }
gfCNCPoint4[26112] = {X 475.6812, Y 92.7038, Z -6.3333, A 0.000, B 0.000, C 0.000 }
gfCNCPoint4[26113] = {X 476.0454, Y 92.7970, Z -6.3333, A 0.000, B 0.000, C 0.000 }
gfCNCPoint4[26114] = {X 476.4049, Y 92.9073, Z -6.3333, A 0.000, B 0.000, C 0.000 }
gfCNCPoint4[26115] = {X 477.2338, Y 93.2831, Z -6.3333, A 0.000, B 0.000, C 0.000 }
gfCNCPoint4[26116] = {X 477.9671, Y 93.8220, Z -6.3333, A 0.000, B 0.000, C 0.000 }
gfCNCPoint4[26117] = {X 478.5731, Y 94.5009, Z -6.3333, A 0.000, B 0.000, C 0.000 }
gfCNCPoint4[26118] = {X 479.0258, Y 95.2905, Z -6.3333, A 0.000, B 0.000, C 0.000 }
gfCNCPoint4[26119] = {X 479.3054, Y 96.1565, Z -6.3333, A 0.000, B 0.000, C 0.000 }
gfCNCPoint4[26120] = {X 479.4000, Y 97.0617, Z -6.3333, A 0.000, B 0.000, C 0.000 }
gfCNCPoint4[26121] = {X 479.4000, Y 97.6951, Z -6.3333, A 0.000, B 0.000, C 0.000 }
gfCNCPoint4[26122] = {X 479.8800, Y 97.6951, Z -6.3333, A 0.000, B 0.000, C 0.000 }
gfCNCPoint4[26123] = {X 507.6813, Y 97.6951, Z -6.3333, A 0.000, B 0.000, C 0.000 }
gfCNCPoint4[26124] = {X 507.6813, Y 100.0951, Z -6.3333, A 0.000, B 0.000, C 0.000 }
gfCNCPoint4[26125] = {X 600.0148, Y 100.0951, Z -6.3333, A 0.000, B 0.000, C 0.000 }
gfCNCPoint4[26126] = {X 600.0672, Y 100.0699, Z -6.3333, A 0.000, B 0.000, C 0.000 }
gfCNCPoint4[26127] = {X 600.0949, Y 100.0187, Z -6.3333, A 0.000, B 0.000, C 0.000 }
gfCNCPoint4[26128] = {X 600.0966, Y 99.1432, Z -6.3333, A 0.000, B 0.000, C 0.000 }
gfCNCPoint4[26129] = {X 600.0966, Y 49.8790, Z -6.3333, A 0.000, B 0.000, C 0.000 }
gfCNCPoint4[26130] = {X 601.1112, Y 49.7518, Z -6.3333, A 0.000, B 0.000, C 0.000 }
gfCNCPoint4[26131] = {X 602.0770, Y 49.4159, Z -6.3333, A 0.000, B 0.000, C 0.000 }
gfCNCPoint4[26132] = {X 602.9516, Y 48.8862, Z -6.3333, A 0.000, B 0.000, C 0.000 }
gfCNCPoint4[26133] = {X 603.6966, Y 48.1858, Z -6.3333, A 0.000, B 0.000, C 0.000 }
gfCNCPoint4[26134] = {X 603.6966, Y 47.3864, Z -6.3333, A 0.000, B 0.000, C 0.000 }
gfCNCPoint4[26135] = {X 603.1147, Y 48.1078, Z -6.3333, A 0.000, B 0.000, C 0.000 }
gfCNCPoint4[26136] = {X 602.3945, Y 48.6914, Z -6.3333, A 0.000, B 0.000, C 0.000 }
gfCNCPoint4[26137] = {X 601.6469, Y 49.0802, Z -6.3333, A 0.000, B 0.000, C 0.000 }
gfCNCPoint4[26138] = {X 600.8388, Y 49.3193, Z -6.3333, A 0.000, B 0.000, C 0.000 }
gfCNCPoint4[26139] = {X 600.0000, Y 49.4000, Z -6.3333, A 0.000, B 0.000, C 0.000 }
gfCNCPoint4[26140] = {X 593.5565, Y 49.4000, Z -6.3333, A 0.000, B 0.000, C 0.000 }
gfCNCPoint4[26141] = {X 592.5988, Y 49.2945, Z -6.3333, A 0.000, B 0.000, C 0.000 }
gfCNCPoint4[26142] = {X 591.6870, Y 48.9831, Z -6.3333, A 0.000, B 0.000, C 0.000 }
gfCNCPoint4[26143] = {X 590.8648, Y 48.4806, Z -6.3333, A 0.000, B 0.000, C 0.000 }
gfCNCPoint4[26144] = {X 590.1717, Y 47.8112, Z -6.3333, A 0.000, B 0.000, C 0.000 }
gfCNCPoint4[26145] = {X 589.6410, Y 47.0071, Z -6.3333, A 0.000, B 0.000, C 0.000 }
gfCNCPoint4[26146] = {X 589.3741, Y 46.3664, Z -6.3333, A 0.000, B 0.000, C 0.000 }
gfCNCPoint4[26147] = {X 589.2113, Y 45.6918, Z -6.3333, A 0.000, B 0.000, C 0.000 }
gfCNCPoint4[26148] = {X 589.1565, Y 45.0000, Z -6.3333, A 0.000, B 0.000, C 0.000 }
gfCNCPoint4[26149] = {X 589.1565, Y 44.0643, Z -6.3333, A 0.000, B 0.000, C 0.000 }
gfCNCPoint4[26150] = {X 589.2604, Y 43.1278, Z -6.3333, A 0.000, B 0.000, C 0.000 }
gfCNCPoint4[26151] = {X 589.5597, Y 42.2344, Z -6.3333, A 0.000, B 0.000, C 0.000 }
gfCNCPoint4[26152] = {X 590.0408, Y 41.4242, Z -6.3333, A 0.000, B 0.000, C 0.000 }
gfCNCPoint4[26153] = {X 590.6821, Y 40.7339, Z -6.3333, A 0.000, B 0.000, C 0.000 }
gfCNCPoint4[26154] = {X 590.6834, Y 40.3069, Z -6.3333, A 0.000, B 0.000, C 0.000 }
gfCNCPoint4[26155] = {X 590.6828, Y 35.2195, Z -6.3333, A 0.000, B 0.000, C 0.000 }
gfCNCPoint4[26156] = {X 590.6826, Y 33.9419, Z -6.3333, A 0.000, B 0.000, C 0.000 }
gfCNCPoint4[26157] = {X 590.2027, Y 35.1260, Z -6.3333, A 0.000, B 0.000, C 0.000 }
gfCNCPoint4[26158] = {X 585.5192, Y 46.6830, Z -6.3333, A 0.000, B 0.000, C 0.000 }
gfCNCPoint4[26159] = {X 585.4476, Y 46.8466, Z -6.3333, A 0.000, B 0.000, C 0.000 }
gfCNCPoint4[26160] = {X 585.3694, Y 47.0071, Z -6.3333, A 0.000, B 0.000, C 0.000 }
gfCNCPoint4[26161] = {X 584.8417, Y 47.8075, Z -6.3333, A 0.000, B 0.000, C 0.000 }
gfCNCPoint4[26162] = {X 584.1532, Y 48.4747, Z -6.3333, A 0.000, B 0.000, C 0.000 }
gfCNCPoint4[26163] = {X 583.3365, Y 48.9769, Z -6.3333, A 0.000, B 0.000, C 0.000 }
gfCNCPoint4[26164] = {X 582.4111, Y 49.2946, Z -6.3333, A 0.000, B 0.000, C 0.000 }
gfCNCPoint4[26165] = {X 581.4384, Y 49.4000, Z -6.3333, A 0.000, B 0.000, C 0.000 }
gfCNCPoint4[26166] = {X 580.4664, Y 49.2878, Z -6.3333, A 0.000, B 0.000, C 0.000 }
gfCNCPoint4[26167] = {X 579.5433, Y 48.9635, Z -6.3333, A 0.000, B 0.000, C 0.000 }
gfCNCPoint4[26168] = {X 578.7146, Y 48.4433, Z -6.3333, A 0.000, B 0.000, C 0.000 }
gfCNCPoint4[26169] = {X 578.0214, Y 47.7529, Z -6.3333, A 0.000, B 0.000, C 0.000 }
gfCNCPoint4[26170] = {X 577.4979, Y 46.9263, Z -6.3333, A 0.000, B 0.000, C 0.000 }
gfCNCPoint4[26171] = {X 577.4375, Y 46.7968, Z -6.3333, A 0.000, B 0.000, C 0.000 }
gfCNCPoint4[26172] = {X 577.3813, Y 46.6655, Z -6.3333, A 0.000, B 0.000, C 0.000 }
gfCNCPoint4[26173] = {X 572.0996, Y 33.7502, Z -6.3333, A 0.000, B 0.000, C 0.000 }
gfCNCPoint4[26174] = {X 572.0998, Y 40.7337, Z -6.3333, A 0.000, B 0.000, C 0.000 }
gfCNCPoint4[26175] = {X 572.7441, Y 41.4228, Z -6.3333, A 0.000, B 0.000, C 0.000 }
gfCNCPoint4[26176] = {X 573.2266, Y 42.2333, Z -6.3333, A 0.000, B 0.000, C 0.000 }
gfCNCPoint4[26177] = {X 573.5253, Y 43.1281, Z -6.3333, A 0.000, B 0.000, C 0.000 }
gfCNCPoint4[26178] = {X 573.6264, Y 44.0660, Z -6.3333, A 0.000, B 0.000, C 0.000 }
gfCNCPoint4[26179] = {X 573.6264, Y 45.0000, Z -6.3333, A 0.000, B 0.000, C 0.000 }
gfCNCPoint4[26180] = {X 573.5140, Y 45.9884, Z -6.3333, A 0.000, B 0.000, C 0.000 }
gfCNCPoint4[26181] = {X 573.1824, Y 46.9263, Z -6.3333, A 0.000, B 0.000, C 0.000 }
gfCNCPoint4[26182] = {X 572.8094, Y 47.5539, Z -6.3333, A 0.000, B 0.000, C 0.000 }
gfCNCPoint4[26183] = {X 572.3377, Y 48.1113, Z -6.3333, A 0.000, B 0.000, C 0.000 }
gfCNCPoint4[26184] = {X 571.6709, Y 48.6585, Z -6.3333, A 0.000, B 0.000, C 0.000 }
gfCNCPoint4[26185] = {X 570.9102, Y 49.0651, Z -6.3333, A 0.000, B 0.000, C 0.000 }
gfCNCPoint4[26186] = {X 570.0848, Y 49.3155, Z -6.3333, A 0.000, B 0.000, C 0.000 }
gfCNCPoint4[26187] = {X 569.2264, Y 49.4000, Z -6.3333, A 0.000, B 0.000, C 0.000 }
gfCNCPoint4[26188] = {X 562.4443, Y 49.4000, Z -6.3333, A 0.000, B 0.000, C 0.000 }
gfCNCPoint4[26189] = {X 561.6617, Y 49.3298, Z -6.3333, A 0.000, B 0.000, C 0.000 }
gfCNCPoint4[26190] = {X 560.9040, Y 49.1216, Z -6.3333, A 0.000, B 0.000, C 0.000 }
gfCNCPoint4[26191] = {X 560.1954, Y 48.7819, Z -6.3333, A 0.000, B 0.000, C 0.000 }
gfCNCPoint4[26192] = {X 559.5586, Y 48.3216, Z -6.3333, A 0.000, B 0.000, C 0.000 }
gfCNCPoint4[26193] = {X 558.9194, Y 47.6334, Z -6.3333, A 0.000, B 0.000, C 0.000 }
gfCNCPoint4[26194] = {X 558.4407, Y 46.8252, Z -6.3333, A 0.000, B 0.000, C 0.000 }
gfCNCPoint4[26195] = {X 558.1446, Y 45.9339, Z -6.3333, A 0.000, B 0.000, C 0.000 }
gfCNCPoint4[26196] = {X 558.0443, Y 45.0000, Z -6.3333, A 0.000, B 0.000, C 0.000 }
gfCNCPoint4[26197] = {X 558.0443, Y 44.0645, Z -6.3333, A 0.000, B 0.000, C 0.000 }
gfCNCPoint4[26198] = {X 558.1479, Y 43.1277, Z -6.3333, A 0.000, B 0.000, C 0.000 }
gfCNCPoint4[26199] = {X 558.4474, Y 42.2340, Z -6.3333, A 0.000, B 0.000, C 0.000 }
gfCNCPoint4[26200] = {X 558.9290, Y 41.4238, Z -6.3333, A 0.000, B 0.000, C 0.000 }
gfCNCPoint4[26201] = {X 559.5712, Y 40.7339, Z -6.3333, A 0.000, B 0.000, C 0.000 }
gfCNCPoint4[26202] = {X 559.5712, Y 9.2665, Z -6.3333, A 0.000, B 0.000, C 0.000 }
gfCNCPoint4[26203] = {X 558.9268, Y 8.5774, Z -6.3333, A 0.000, B 0.000, C 0.000 }
gfCNCPoint4[26204] = {X 558.4442, Y 7.7668, Z -6.3333, A 0.000, B 0.000, C 0.000 }
gfCNCPoint4[26205] = {X 558.1454, Y 6.8720, Z -6.3333, A 0.000, B 0.000, C 0.000 }
gfCNCPoint4[26206] = {X 558.0443, Y 5.9340, Z -6.3333, A 0.000, B 0.000, C 0.000 }
gfCNCPoint4[26207] = {X 558.0443, Y 5.0000, Z -6.3333, A 0.000, B 0.000, C 0.000 }
gfCNCPoint4[26208] = {X 558.1353, Y 4.1096, Z -6.3333, A 0.000, B 0.000, C 0.000 }
gfCNCPoint4[26209] = {X 558.4046, Y 3.2561, Z -6.3333, A 0.000, B 0.000, C 0.000 }
gfCNCPoint4[26210] = {X 558.9155, Y 2.3717, Z -6.3333, A 0.000, B 0.000, C 0.000 }
gfCNCPoint4[26211] = {X 559.6166, Y 1.6289, Z -6.3333, A 0.000, B 0.000, C 0.000 }
gfCNCPoint4[26212] = {X 560.4700, Y 1.0678, Z -6.3333, A 0.000, B 0.000, C 0.000 }
gfCNCPoint4[26213] = {X 561.4298, Y 0.7185, Z -6.3333, A 0.000, B 0.000, C 0.000 }
gfCNCPoint4[26214] = {X 562.4443, Y 0.6000, Z -6.3333, A 0.000, B 0.000, C 0.000 }
gfCNCPoint4[26215] = {X 570.9376, Y 0.6000, Z -6.3333, A 0.000, B 0.000, C 0.000 }
gfCNCPoint4[26216] = {X 571.9520, Y 0.7185, Z -6.3333, A 0.000, B 0.000, C 0.000 }
gfCNCPoint4[26217] = {X 572.9118, Y 1.0678, Z -6.3333, A 0.000, B 0.000, C 0.000 }
gfCNCPoint4[26218] = {X 573.7653, Y 1.6289, Z -6.3333, A 0.000, B 0.000, C 0.000 }
gfCNCPoint4[26219] = {X 574.4663, Y 2.3717, Z -6.3333, A 0.000, B 0.000, C 0.000 }
gfCNCPoint4[26220] = {X 574.9772, Y 3.2561, Z -6.3333, A 0.000, B 0.000, C 0.000 }
gfCNCPoint4[26221] = {X 575.2317, Y 4.0406, Z -6.3333, A 0.000, B 0.000, C 0.000 }
gfCNCPoint4[26222] = {X 575.3353, Y 4.8589, Z -6.3333, A 0.000, B 0.000, C 0.000 }
gfCNCPoint4[26223] = {X 580.1328, Y 4.7049, Z -6.3333, A 0.000, B 0.000, C 0.000 }
gfCNCPoint4[26224] = {X 580.1364, Y 4.8524, Z -6.3333, A 0.000, B 0.000, C 0.000 }
gfCNCPoint4[26225] = {X 580.1376, Y 5.0000, Z -6.3333, A 0.000, B 0.000, C 0.000 }
gfCNCPoint4[26226] = {X 580.1368, Y 6.0531, Z -6.3333, A 0.000, B 0.000, C 0.000 }
gfCNCPoint4[26227] = {X 580.0609, Y 7.1189, Z -6.3333, A 0.000, B 0.000, C 0.000 }
gfCNCPoint4[26228] = {X 579.8620, Y 8.1688, Z -6.3333, A 0.000, B 0.000, C 0.000 }
gfCNCPoint4[26229] = {X 581.1999, Y 11.4531, Z -6.3333, A 0.000, B 0.000, C 0.000 }
gfCNCPoint4[26230] = {X 582.6183, Y 7.9842, Z -6.3333, A 0.000, B 0.000, C 0.000 }
gfCNCPoint4[26231] = {X 582.4488, Y 6.9994, Z -6.3333, A 0.000, B 0.000, C 0.000 }
gfCNCPoint4[26232] = {X 582.3872, Y 6.0021, Z -6.3333, A 0.000, B 0.000, C 0.000 }
gfCNCPoint4[26233] = {X 582.3870, Y 5.0000, Z -6.3333, A 0.000, B 0.000, C 0.000 }
gfCNCPoint4[26234] = {X 582.3881, Y 4.8524, Z -6.3333, A 0.000, B 0.000, C 0.000 }
gfCNCPoint4[26235] = {X 582.3917, Y 4.7049, Z -6.3333, A 0.000, B 0.000, C 0.000 }
gfCNCPoint4[26236] = {X 580.1328, Y 4.7049, Z -6.3333, A 0.000, B 0.000, C 0.000 }
gfCNCPoint4[26237] = {X 577.7341, Y 4.7819, Z -6.3333, A 0.000, B 0.000, C 0.000 }
gfCNCPoint4[26238] = {X 577.7367, Y 4.8909, Z -6.3333, A 0.000, B 0.000, C 0.000 }
gfCNCPoint4[26239] = {X 577.7376, Y 5.0000, Z -6.3333, A 0.000, B 0.000, C 0.000 }
gfCNCPoint4[26240] = {X 577.7370, Y 6.0220, Z -6.3333, A 0.000, B 0.000, C 0.000 }
gfCNCPoint4[26241] = {X 577.6240, Y 7.1716, Z -6.3333, A 0.000, B 0.000, C 0.000 }
gfCNCPoint4[26242] = {X 577.3180, Y 8.2855, Z -6.3333, A 0.000, B 0.000, C 0.000 }
gfCNCPoint4[26243] = {X 581.1958, Y 17.8045, Z -6.3333, A 0.000, B 0.000, C 0.000 }
gfCNCPoint4[26244] = {X 585.1514, Y 8.1303, Z -6.3333, A 0.000, B 0.000, C 0.000 }
gfCNCPoint4[26245] = {X 584.8835, Y 7.0756, Z -6.3333, A 0.000, B 0.000, C 0.000 }
gfCNCPoint4[26246] = {X 584.7872, Y 5.9916, Z -6.3333, A 0.000, B 0.000, C 0.000 }
gfCNCPoint4[26247] = {X 584.7870, Y 5.0000, Z -6.3333, A 0.000, B 0.000, C 0.000 }
gfCNCPoint4[26248] = {X 584.7878, Y 4.8909, Z -6.3333, A 0.000, B 0.000, C 0.000 }
gfCNCPoint4[26249] = {X 584.7905, Y 4.7819, Z -6.3333, A 0.000, B 0.000, C 0.000 }
gfCNCPoint4[26250] = {X 584.9506, Y 3.5173, Z -6.3333, A 0.000, B 0.000, C 0.000 }
gfCNCPoint4[26251] = {X 585.3438, Y 2.3049, Z -6.3333, A 0.000, B 0.000, C 0.000 }
gfCNCPoint4[26252] = {X 577.1807, Y 2.3049, Z -6.3333, A 0.000, B 0.000, C 0.000 }
gfCNCPoint4[26253] = {X 577.5739, Y 3.5173, Z -6.3333, A 0.000, B 0.000, C 0.000 }
gfCNCPoint4[26254] = {X 577.7341, Y 4.7819, Z -6.3333, A 0.000, B 0.000, C 0.000 }
gfCNCPoint4[26255] = {X 575.3353, Y 4.8589, Z -6.3333, A 0.000, B 0.000, C 0.000 }
gfCNCPoint4[26256] = {X 575.3370, Y 4.9294, Z -6.3333, A 0.000, B 0.000, C 0.000 }
gfCNCPoint4[26257] = {X 575.3376, Y 5.0000, Z -6.3333, A 0.000, B 0.000, C 0.000 }
gfCNCPoint4[26258] = {X 575.3372, Y 5.9910, Z -6.3333, A 0.000, B 0.000, C 0.000 }
gfCNCPoint4[26259] = {X 575.2577, Y 6.7685, Z -6.3333, A 0.000, B 0.000, C 0.000 }
gfCNCPoint4[26260] = {X 575.0419, Y 7.5197, Z -6.3333, A 0.000, B 0.000, C 0.000 }
gfCNCPoint4[26261] = {X 574.6967, Y 8.2208, Z -6.3333, A 0.000, B 0.000, C 0.000 }
gfCNCPoint4[26262] = {X 575.2866, Y 9.6563, Z -6.3333, A 0.000, B 0.000, C 0.000 }
gfCNCPoint4[26263] = {X 578.9730, Y 18.7096, Z -6.3333, A 0.000, B 0.000, C 0.000 }
gfCNCPoint4[26264] = {X 580.9325, Y 23.5217, Z -6.3333, A 0.000, B 0.000, C 0.000 }
gfCNCPoint4[26265] = {X 581.1912, Y 24.1571, Z -6.3333, A 0.000, B 0.000, C 0.000 }
gfCNCPoint4[26266] = {X 587.7568, Y 8.0997, Z -6.3333, A 0.000, B 0.000, C 0.000 }
gfCNCPoint4[26267] = {X 587.4433, Y 7.4141, Z -6.3333, A 0.000, B 0.000, C 0.000 }
gfCNCPoint4[26268] = {X 587.2515, Y 6.6851, Z -6.3333, A 0.000, B 0.000, C 0.000 }
gfCNCPoint4[26269] = {X 587.1870, Y 5.9340, Z -6.3333, A 0.000, B 0.000, C 0.000 }
gfCNCPoint4[26270] = {X 587.1870, Y 5.0000, Z -6.3333, A 0.000, B 0.000, C 0.000 }
gfCNCPoint4[26271] = {X 587.2780, Y 4.1096, Z -6.3333, A 0.000, B 0.000, C 0.000 }
gfCNCPoint4[26272] = {X 587.5473, Y 3.2561, Z -6.3333, A 0.000, B 0.000, C 0.000 }
gfCNCPoint4[26273] = {X 588.0582, Y 2.3717, Z -6.3333, A 0.000, B 0.000, C 0.000 }
gfCNCPoint4[26274] = {X 588.7593, Y 1.6289, Z -6.3333, A 0.000, B 0.000, C 0.000 }
gfCNCPoint4[26275] = {X 589.6127, Y 1.0678, Z -6.3333, A 0.000, B 0.000, C 0.000 }
gfCNCPoint4[26276] = {X 590.5725, Y 0.7185, Z -6.3333, A 0.000, B 0.000, C 0.000 }
gfCNCPoint4[26277] = {X 591.5870, Y 0.6000, Z -6.3333, A 0.000, B 0.000, C 0.000 }
gfCNCPoint4[26278] = {X 600.0000, Y 0.6000, Z -6.3333, A 0.000, B 0.000, C 0.000 }
gfCNCPoint4[26279] = {X 600.8720, Y 0.6873, Z -6.3333, A 0.000, B 0.000, C 0.000 }
gfCNCPoint4[26280] = {X 601.7095, Y 0.9457, Z -6.3333, A 0.000, B 0.000, C 0.000 }
gfCNCPoint4[26281] = {X 602.4791, Y 1.3649, Z -6.3333, A 0.000, B 0.000, C 0.000 }
gfCNCPoint4[26282] = {X 603.1504, Y 1.9283, Z -6.3333, A 0.000, B 0.000, C 0.000 }
gfCNCPoint4[26283] = {X 603.6966, Y 2.6136, Z -6.3333, A 0.000, B 0.000, C 0.000 }
gfCNCPoint4[26284] = {X 603.6966, Y 1.8142, Z -6.3333, A 0.000, B 0.000, C 0.000 }
gfCNCPoint4[26285] = {X 602.9513, Y 1.1136, Z -6.3333, A 0.000, B 0.000, C 0.000 }
gfCNCPoint4[26286] = {X 602.0764, Y 0.5838, Z -6.3333, A 0.000, B 0.000, C 0.000 }
gfCNCPoint4[26287] = {X 601.1102, Y 0.2480, Z -6.3333, A 0.000, B 0.000, C 0.000 }
gfCNCPoint4[26288] = {X 600.0952, Y 0.1209, Z -6.3333, A 0.000, B 0.000, C 0.000 }
gfCNCPoint4[26289] = {X 600.0949, Y -0.0187, Z -6.3333, A 0.000, B 0.000, C 0.000 }
gfCNCPoint4[26290] = {X 600.0672, Y -0.0699, Z -6.3333, A 0.000, B 0.000, C 0.000 }
gfCNCPoint4[26291] = {X 600.0148, Y -0.0951, Z -6.3333, A 0.000, B 0.000, C 0.000 }
gfCNCPoint4[26292] = {X 351.5685, Y -0.0951, Z -6.3333, A 0.000, B 0.000, C 0.000 }
gfCNCPoint4[26293] = {X 351.4213, Y -0.1227, Z -6.3333, A 0.000, B 0.000, C 0.000 }
gfCNCPoint4[26294] = {X 348.9218, Y -0.4705, Z -6.3333, A 0.000, B 0.000, C 0.000 }
gfCNCPoint4[26295] = {X 346.4007, Y -0.5821, Z -6.3333, A 0.000, B 0.000, C 0.000 }
gfCNCPoint4[26296] = {X 343.8802, Y -0.4566, Z -6.3333, A 0.000, B 0.000, C 0.000 }
gfCNCPoint4[26297] = {X 341.3827, Y -0.0951, Z -6.3333, A 0.000, B 0.000, C 0.000 }
gfCNCPoint4[26298] = {X -0.0148, Y -0.0951, Z -6.3333, A 0.000, B 0.000, C 0.000 }
gfCNCPoint4[26299] = {X -0.0672, Y -0.0699, Z -6.3333, A 0.000, B 0.000, C 0.000 }
gfCNCPoint4[26300] = {X -0.0949, Y -0.0187, Z -6.3333, A 0.000, B 0.000, C 0.000 }
gfCNCPoint4[26301] = {X -0.0966, Y 0.8568, Z -6.3333, A 0.000, B 0.000, C 0.000 }
gfCNCPoint4[26302] = {X -0.0966, Y 8.7891, Z -6.3333, A 0.000, B 0.000, C 0.000 }
gfCNCPoint4[26303] = {X -0.7634, Y 8.9979, Z -6.3333, A 0.000, B 0.000, C 0.000 }
gfCNCPoint4[26304] = {X -1.3934, Y 9.2998, Z -6.3333, A 0.000, B 0.000, C 0.000 }
gfCNCPoint4[26305] = {X -1.9904, Y 9.6404, Z -6.3333, A 0.000, B 0.000, C 0.000 }
gfCNCPoint4[26306] = {X -2.6455, Y 10.0884, Z -6.3333, A 0.000, B 0.000, C 0.000 }
gfCNCPoint4[26307] = {X -3.2193, Y 10.6367, Z -6.3333, A 0.000, B 0.000, C 0.000 }
gfCNCPoint4[26308] = {X -3.6966, Y 11.2708, Z -6.3333, A 0.000, B 0.000, C 0.000 }
gfCNCPoint4[26309] = {X -3.6966, Y 12.3464, Z -6.3333, A 0.000, B 0.000, C 0.000 }
gfCNCPoint4[26310] = {X -3.2333, Y 11.4385, Z -6.3333, A 0.000, B 0.000, C 0.000 }
gfCNCPoint4[26311] = {X -2.5735, Y 10.6616, Z -6.3333, A 0.000, B 0.000, C 0.000 }
gfCNCPoint4[26312] = {X -1.7526, Y 10.0573, Z -6.3333, A 0.000, B 0.000, C 0.000 }
gfCNCPoint4[26313] = {X -1.0994, Y 9.6852, Z -6.3333, A 0.000, B 0.000, C 0.000 }
gfCNCPoint4[26314] = {X -0.1608, Y 9.3012, Z -6.3333, A 0.000, B 0.000, C 0.000 }
gfCNCPoint4[26315] = {X 0.8408, Y 9.1423, Z -6.3333, A 0.000, B 0.000, C 0.000 }
gfCNCPoint4[26316] = {X 1.8521, Y 9.2169, Z -6.3333, A 0.000, B 0.000, C 0.000 }
gfCNCPoint4[26317] = {X 2.2305, Y 9.3069, Z -6.3333, A 0.000, B 0.000, C 0.000 }
gfCNCPoint4[26318] = {X 2.5995, Y 9.4299, Z -6.3333, A 0.000, B 0.000, C 0.000 }
gfCNCPoint4[26319] = {X 3.4586, Y 9.0456, Z -6.3333, A 0.000, B 0.000, C 0.000 }
gfCNCPoint4[26320] = {X 5.5422, Y 8.2606, Z -6.3333, A 0.000, B 0.000, C 0.000 }
gfCNCPoint4[26321] = {X 7.6900, Y 7.6731, Z -6.3333, A 0.000, B 0.000, C 0.000 }
gfCNCPoint4[26322] = {X 9.8831, Y 7.2882, Z -6.3333, A 0.000, B 0.000, C 0.000 }
gfCNCPoint4[26323] = {X 12.1025, Y 7.1091, Z -6.3333, A 0.000, B 0.000, C 0.000 }
gfCNCPoint4[26324] = {X 14.3290, Y 7.1376, Z -6.3333, A 0.000, B 0.000, C 0.000 }
gfCNCPoint4[26325] = {X 16.5431, Y 7.3732, Z -6.3333, A 0.000, B 0.000, C 0.000 }
gfCNCPoint4[26326] = {X 18.2868, Y 7.7304, Z -6.3333, A 0.000, B 0.000, C 0.000 }
gfCNCPoint4[26327] = {X 19.9852, Y 8.2625, Z -6.3333, A 0.000, B 0.000, C 0.000 }
gfCNCPoint4[26328] = {X 21.6210, Y 8.9642, Z -6.3333, A 0.000, B 0.000, C 0.000 }
gfCNCPoint4[26329] = {X 23.1771, Y 9.8281, Z -6.3333, A 0.000, B 0.000, C 0.000 }
gfCNCPoint4[26330] = {X 24.6376, Y 10.8454, Z -6.3333, A 0.000, B 0.000, C 0.000 }
gfCNCPoint4[26331] = {X 25.7302, Y 11.8009, Z -6.3333, A 0.000, B 0.000, C 0.000 }
gfCNCPoint4[26332] = {X 26.7101, Y 12.8716, Z -6.3333, A 0.000, B 0.000, C 0.000 }
gfCNCPoint4[26333] = {X 27.5655, Y 14.0443, Z -6.3333, A 0.000, B 0.000, C 0.000 }
gfCNCPoint4[26334] = {X 28.2856, Y 15.3045, Z -6.3333, A 0.000, B 0.000, C 0.000 }
gfCNCPoint4[26335] = {X 28.8617, Y 16.6367, Z -6.3333, A 0.000, B 0.000, C 0.000 }
gfCNCPoint4[26336] = {X 29.3385, Y 18.3012, Z -6.3333, A 0.000, B 0.000, C 0.000 }
gfCNCPoint4[26337] = {X 29.6214, Y 20.0093, Z -6.3333, A 0.000, B 0.000, C 0.000 }
gfCNCPoint4[26338] = {X 29.7066, Y 21.7387, Z -6.3333, A 0.000, B 0.000, C 0.000 }
gfCNCPoint4[26339] = {X 29.5930, Y 23.4664, Z -6.3333, A 0.000, B 0.000, C 0.000 }
gfCNCPoint4[26340] = {X 29.2821, Y 25.1697, Z -6.3333, A 0.000, B 0.000, C 0.000 }
gfCNCPoint4[26341] = {X 28.7906, Y 26.7455, Z -6.3333, A 0.000, B 0.000, C 0.000 }
gfCNCPoint4[26342] = {X 28.0836, Y 28.2371, Z -6.3333, A 0.000, B 0.000, C 0.000 }
gfCNCPoint4[26343] = {X 27.1749, Y 29.6152, Z -6.3333, A 0.000, B 0.000, C 0.000 }
gfCNCPoint4[26344] = {X 26.3578, Y 30.5723, Z -6.3333, A 0.000, B 0.000, C 0.000 }
gfCNCPoint4[26345] = {X 25.4433, Y 31.4367, Z -6.3333, A 0.000, B 0.000, C 0.000 }
gfCNCPoint4[26346] = {X 26.1252, Y 31.7405, Z -6.3333, A 0.000, B 0.000, C 0.000 }
gfCNCPoint4[26347] = {X 26.7460, Y 32.1552, Z -6.3333, A 0.000, B 0.000, C 0.000 }
gfCNCPoint4[26348] = {X 27.2878, Y 32.6689, Z -6.3333, A 0.000, B 0.000, C 0.000 }
gfCNCPoint4[26349] = {X 27.6592, Y 33.1494, Z -6.3333, A 0.000, B 0.000, C 0.000 }
gfCNCPoint4[26350] = {X 27.9609, Y 33.6765, Z -6.3333, A 0.000, B 0.000, C 0.000 }
gfCNCPoint4[26351] = {X 30.9820, Y 39.9182, Z -6.3333, A 0.000, B 0.000, C 0.000 }
gfCNCPoint4[26352] = {X 31.3085, Y 40.8441, Z -6.3333, A 0.000, B 0.000, C 0.000 }
gfCNCPoint4[26353] = {X 31.4215, Y 41.8194, Z -6.3333, A 0.000, B 0.000, C 0.000 }
gfCNCPoint4[26354] = {X 31.3155, Y 42.7955, Z -6.3333, A 0.000, B 0.000, C 0.000 }
gfCNCPoint4[26355] = {X 30.9956, Y 43.7238, Z -6.3333, A 0.000, B 0.000, C 0.000 }
gfCNCPoint4[26356] = {X 30.4779, Y 44.5580, Z -6.3333, A 0.000, B 0.000, C 0.000 }
gfCNCPoint4[26357] = {X 29.7880, Y 45.2567, Z -6.3333, A 0.000, B 0.000, C 0.000 }
gfCNCPoint4[26358] = {X 29.2520, Y 45.6901, Z -6.3333, A 0.000, B 0.000, C 0.000 }
gfCNCPoint4[26359] = {X 28.5411, Y 46.1591, Z -6.3333, A 0.000, B 0.000, C 0.000 }
gfCNCPoint4[26360] = {X 27.7535, Y 46.4828, Z -6.3333, A 0.000, B 0.000, C 0.000 }
gfCNCPoint4[26361] = {X 26.9182, Y 46.6491, Z -6.3333, A 0.000, B 0.000, C 0.000 }
gfCNCPoint4[26362] = {X 26.0666, Y 46.6519, Z -6.3333, A 0.000, B 0.000, C 0.000 }
gfCNCPoint4[26363] = {X 25.2304, Y 46.4909, Z -6.3333, A 0.000, B 0.000, C 0.000 }
gfCNCPoint4[26364] = {X 23.4342, Y 47.4359, Z -6.3333, A 0.000, B 0.000, C 0.000 }
gfCNCPoint4[26365] = {X 21.5772, Y 48.2549, Z -6.3333, A 0.000, B 0.000, C 0.000 }
gfCNCPoint4[26366] = {X 19.6682, Y 48.9440, Z -6.3333, A 0.000, B 0.000, C 0.000 }
gfCNCPoint4[26367] = {X 17.7216, Y 49.4935, Z -6.3333, A 0.000, B 0.000, C 0.000 }
gfCNCPoint4[26368] = {X 15.7341, Y 49.8685, Z -6.3333, A 0.000, B 0.000, C 0.000 }
gfCNCPoint4[26369] = {X 13.7211, Y 50.0662, Z -6.3333, A 0.000, B 0.000, C 0.000 }
gfCNCPoint4[26370] = {X 11.6986, Y 50.0850, Z -6.3333, A 0.000, B 0.000, C 0.000 }
gfCNCPoint4[26371] = {X 9.6824, Y 49.9247, Z -6.3333, A 0.000, B 0.000, C 0.000 }
gfCNCPoint4[26372] = {X 7.6882, Y 49.5865, Z -6.3333, A 0.000, B 0.000, C 0.000 }
gfCNCPoint4[26373] = {X 6.2182, Y 49.2053, Z -6.3333, A 0.000, B 0.000, C 0.000 }
gfCNCPoint4[26374] = {X 4.7886, Y 48.6930, Z -6.3333, A 0.000, B 0.000, C 0.000 }
gfCNCPoint4[26375] = {X 3.4112, Y 48.0536, Z -6.3333, A 0.000, B 0.000, C 0.000 }
gfCNCPoint4[26376] = {X 1.9574, Y 47.2019, Z -6.3333, A 0.000, B 0.000, C 0.000 }
gfCNCPoint4[26377] = {X 0.5963, Y 46.2089, Z -6.3333, A 0.000, B 0.000, C 0.000 }
gfCNCPoint4[26378] = {X -0.5427, Y 45.1848, Z -6.3333, A 0.000, B 0.000, C 0.000 }
gfCNCPoint4[26379] = {X -1.5544, Y 44.0347, Z -6.3333, A 0.000, B 0.000, C 0.000 }
gfCNCPoint4[26380] = {X -2.4249, Y 42.7743, Z -6.3333, A 0.000, B 0.000, C 0.000 }
gfCNCPoint4[26381] = {X -3.1422, Y 41.4210, Z -6.3333, A 0.000, B 0.000, C 0.000 }
gfCNCPoint4[26382] = {X -3.6966, Y 39.9931, Z -6.3333, A 0.000, B 0.000, C 0.000 }
gfCNCPoint4[26383] = {X -3.6966, Y 41.3553, Z -6.3333, A 0.000, B 0.000, C 0.000 }
gfCNCPoint4[26384] = {X -3.0107, Y 42.7260, Z -6.3333, A 0.000, B 0.000, C 0.000 }
gfCNCPoint4[26385] = {X -2.1747, Y 44.0106, Z -6.3333, A 0.000, B 0.000, C 0.000 }
gfCNCPoint4[26386] = {X -1.1992, Y 45.1928, Z -6.3333, A 0.000, B 0.000, C 0.000 }
gfCNCPoint4[26387] = {X -0.0966, Y 46.2576, Z -6.3333, A 0.000, B 0.000, C 0.000 }
gfCNCPoint4[26388] = {X -0.0966, Y 99.1432, Z -6.3333, A 0.000, B 0.000, C 0.000 }
